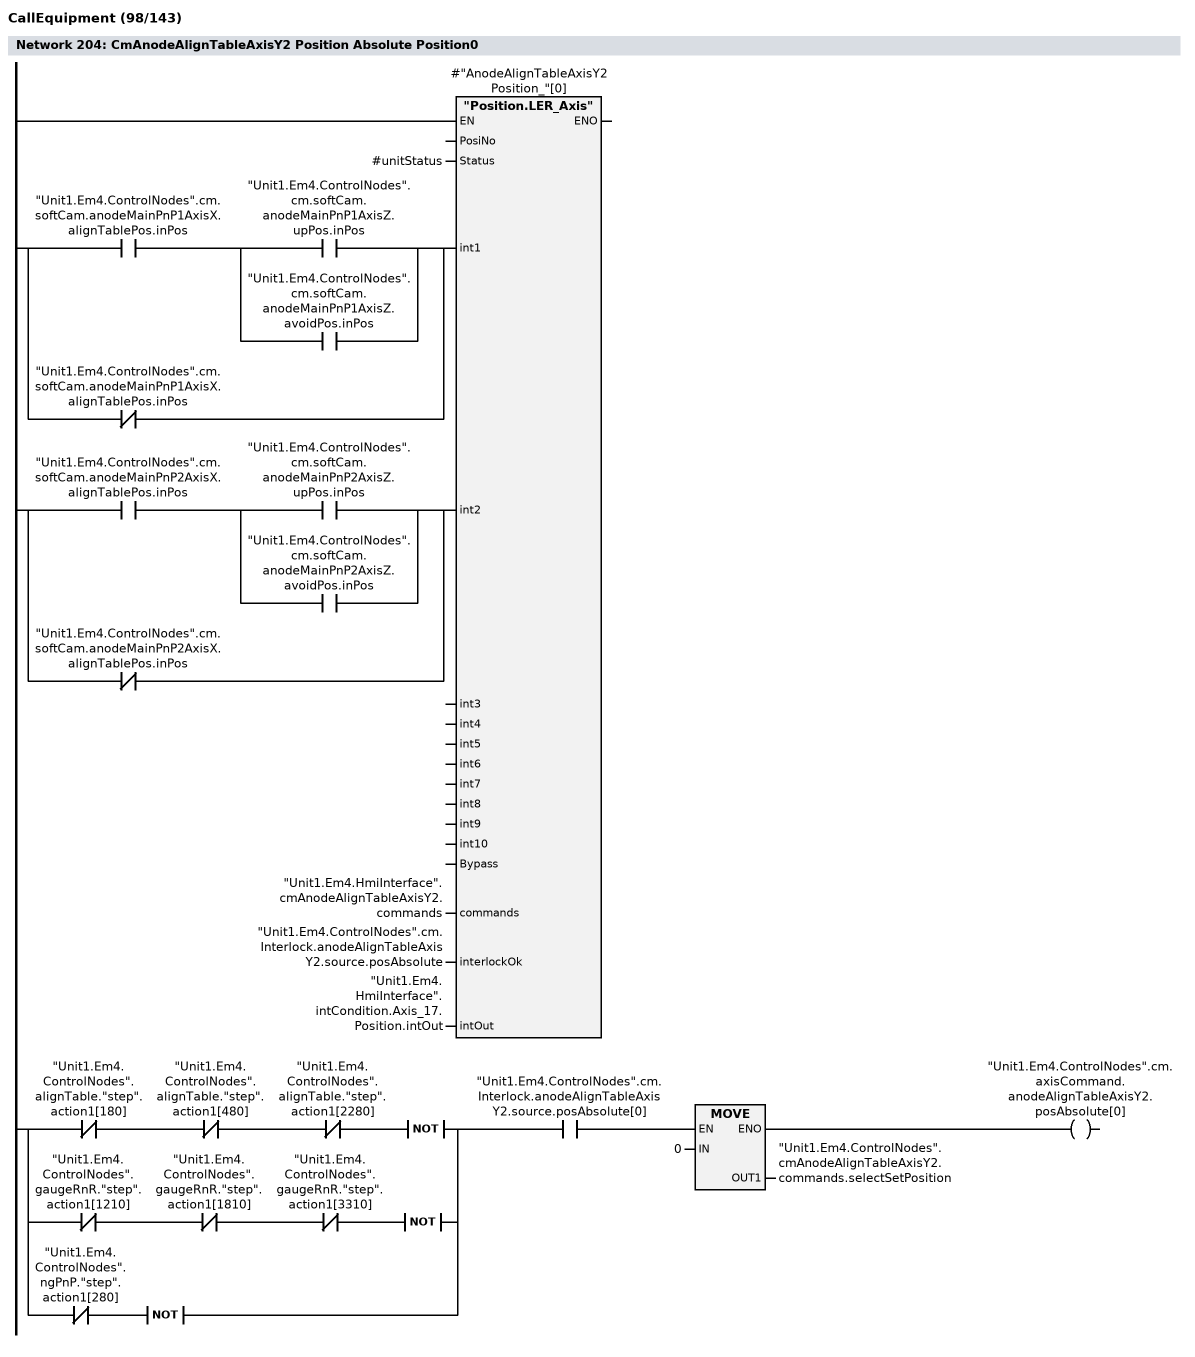
   RUNG wire#powerrail
      #"AnodeAlignTableAxisY2 Position_"[0](int1 := wire#w2, int2 := wire#w4, PosiNo :=, Status := #unitStatus, int3 :=, int4 :=, int5 :=, int6 :=, int7 :=, int8 :=, int9 :=, int10 :=, Bypass :=, commands := "Unit1.Em4.HmiInterface".cmAnodeAlignTableAxisY2.commands, interlockOk := "Unit1.Em4.ControlNodes".cm.Interlock.anodeAlignTableAxisY2.source.posAbsolute, intOut := "Unit1.Em4.HmiInterface".intCondition.Axis_17.Position.intOut)
   END_RUNG
   RUNG wire#powerrail
      Contact( "Unit1.Em4.ControlNodes".cm.softCam.anodeMainPnP1AxisX.alignTablePos.inPos )
      wire#w1
      Contact( "Unit1.Em4.ControlNodes".cm.softCam.anodeMainPnP1AxisZ.upPos.inPos )
   END_RUNG wire#w2
   RUNG wire#w1
      Contact( "Unit1.Em4.ControlNodes".cm.softCam.anodeMainPnP1AxisZ.avoidPos.inPos )
   END_RUNG wire#w2
   RUNG wire#powerrail
      I_Contact( "Unit1.Em4.ControlNodes".cm.softCam.anodeMainPnP1AxisX.alignTablePos.inPos )
   END_RUNG wire#w2
   RUNG wire#powerrail
      Contact( "Unit1.Em4.ControlNodes".cm.softCam.anodeMainPnP2AxisX.alignTablePos.inPos )
      wire#w3
      Contact( "Unit1.Em4.ControlNodes".cm.softCam.anodeMainPnP2AxisZ.upPos.inPos )
   END_RUNG wire#w4
   RUNG wire#w3
      Contact( "Unit1.Em4.ControlNodes".cm.softCam.anodeMainPnP2AxisZ.avoidPos.inPos )
   END_RUNG wire#w4
   RUNG wire#powerrail
      I_Contact( "Unit1.Em4.ControlNodes".cm.softCam.anodeMainPnP2AxisX.alignTablePos.inPos )
   END_RUNG wire#w4
   RUNG wire#powerrail
      I_Contact( "Unit1.Em4.ControlNodes".alignTable."step".action1[180] )
      I_Contact( "Unit1.Em4.ControlNodes".alignTable."step".action1[480] )
      I_Contact( "Unit1.Em4.ControlNodes".alignTable."step".action1[2280] )
      Not()
      wire#w5
      Contact( "Unit1.Em4.ControlNodes".cm.Interlock.anodeAlignTableAxisY2.source.posAbsolute[0] )
      Move(in := 0, out1 => "Unit1.Em4.ControlNodes".cmAnodeAlignTableAxisY2.commands.selectSetPosition)
      Coil( "Unit1.Em4.ControlNodes".cm.axisCommand.anodeAlignTableAxisY2.posAbsolute[0] )
   END_RUNG
   RUNG wire#powerrail
      I_Contact( "Unit1.Em4.ControlNodes".gaugeRnR."step".action1[1210] )
      I_Contact( "Unit1.Em4.ControlNodes".gaugeRnR."step".action1[1810] )
      I_Contact( "Unit1.Em4.ControlNodes".gaugeRnR."step".action1[3310] )
      Not()
   END_RUNG wire#w5
   RUNG wire#powerrail
      I_Contact( "Unit1.Em4.ControlNodes".ngPnP."step".action1[280] )
      Not()
   END_RUNG wire#w5
   // the same network as SCL:
   #"AnodeAlignTableAxisY2 Position_"[0](Status := #unitStatus,   // "Position.LER_Axis"
                           int1 := ("Unit1.Em4.ControlNodes".cm.softCam.anodeMainPnP1AxisX.alignTablePos.inPos AND ("Unit1.Em4.ControlNodes".cm.softCam.anodeMainPnP1AxisZ.upPos.inPos OR "Unit1.Em4.ControlNodes".cm.softCam.anodeMainPnP1AxisZ.avoidPos.inPos)) OR NOT "Unit1.Em4.ControlNodes".cm.softCam.anodeMainPnP1AxisX.alignTablePos.inPos,
                           int2 := ("Unit1.Em4.ControlNodes".cm.softCam.anodeMainPnP2AxisX.alignTablePos.inPos AND ("Unit1.Em4.ControlNodes".cm.softCam.anodeMainPnP2AxisZ.upPos.inPos OR "Unit1.Em4.ControlNodes".cm.softCam.anodeMainPnP2AxisZ.avoidPos.inPos)) OR NOT "Unit1.Em4.ControlNodes".cm.softCam.anodeMainPnP2AxisX.alignTablePos.inPos,
                           commands := "Unit1.Em4.HmiInterface".cmAnodeAlignTableAxisY2.commands,
                           interlockOk := "Unit1.Em4.ControlNodes".cm.Interlock.anodeAlignTableAxisY2.source.posAbsolute,
                           intOut := "Unit1.Em4.HmiInterface".intCondition.Axis_17.Position.intOut);
   #_w1 := (NOT (NOT "Unit1.Em4.ControlNodes".alignTable."step".action1[180] AND NOT "Unit1.Em4.ControlNodes".alignTable."step".action1[480] AND NOT "Unit1.Em4.ControlNodes".alignTable."step".action1[2280]) OR NOT (NOT "Unit1.Em4.ControlNodes".gaugeRnR."step".action1[1210] AND NOT "Unit1.Em4.ControlNodes".gaugeRnR."step".action1[1810] AND NOT "Unit1.Em4.ControlNodes".gaugeRnR."step".action1[3310]) OR NOT (NOT "Unit1.Em4.ControlNodes".ngPnP."step".action1[280])) AND "Unit1.Em4.ControlNodes".cm.Interlock.anodeAlignTableAxisY2.source.posAbsolute[0];
   IF #_w1 THEN "Unit1.Em4.ControlNodes".cmAnodeAlignTableAxisY2.commands.selectSetPosition := 0; END_IF;
   "Unit1.Em4.ControlNodes".cm.axisCommand.anodeAlignTableAxisY2.posAbsolute[0] := #_w1;
END_REGION

REGION Network 205: CmAnodeAlignTableAxisY2 Position Absolute Position1
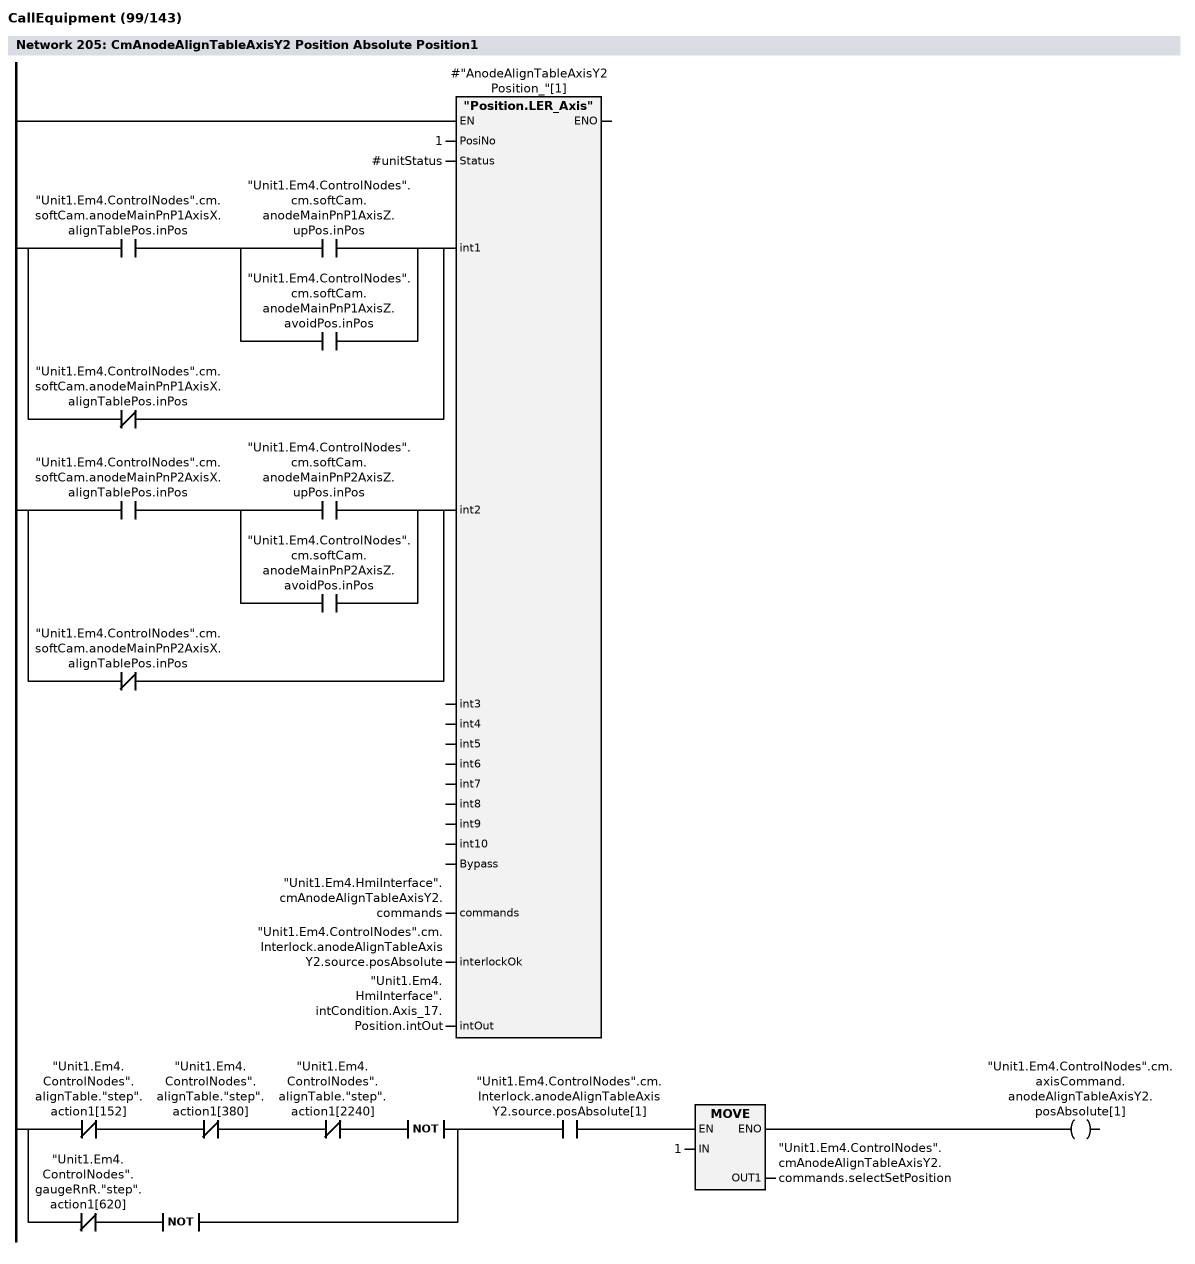
   RUNG wire#powerrail
      #"AnodeAlignTableAxisY2 Position_"[1](int1 := wire#w2, int2 := wire#w4, PosiNo := 1, Status := #unitStatus, int3 :=, int4 :=, int5 :=, int6 :=, int7 :=, int8 :=, int9 :=, int10 :=, Bypass :=, commands := "Unit1.Em4.HmiInterface".cmAnodeAlignTableAxisY2.commands, interlockOk := "Unit1.Em4.ControlNodes".cm.Interlock.anodeAlignTableAxisY2.source.posAbsolute, intOut := "Unit1.Em4.HmiInterface".intCondition.Axis_17.Position.intOut)
   END_RUNG
   RUNG wire#powerrail
      Contact( "Unit1.Em4.ControlNodes".cm.softCam.anodeMainPnP1AxisX.alignTablePos.inPos )
      wire#w1
      Contact( "Unit1.Em4.ControlNodes".cm.softCam.anodeMainPnP1AxisZ.upPos.inPos )
   END_RUNG wire#w2
   RUNG wire#w1
      Contact( "Unit1.Em4.ControlNodes".cm.softCam.anodeMainPnP1AxisZ.avoidPos.inPos )
   END_RUNG wire#w2
   RUNG wire#powerrail
      I_Contact( "Unit1.Em4.ControlNodes".cm.softCam.anodeMainPnP1AxisX.alignTablePos.inPos )
   END_RUNG wire#w2
   RUNG wire#powerrail
      Contact( "Unit1.Em4.ControlNodes".cm.softCam.anodeMainPnP2AxisX.alignTablePos.inPos )
      wire#w3
      Contact( "Unit1.Em4.ControlNodes".cm.softCam.anodeMainPnP2AxisZ.upPos.inPos )
   END_RUNG wire#w4
   RUNG wire#w3
      Contact( "Unit1.Em4.ControlNodes".cm.softCam.anodeMainPnP2AxisZ.avoidPos.inPos )
   END_RUNG wire#w4
   RUNG wire#powerrail
      I_Contact( "Unit1.Em4.ControlNodes".cm.softCam.anodeMainPnP2AxisX.alignTablePos.inPos )
   END_RUNG wire#w4
   RUNG wire#powerrail
      I_Contact( "Unit1.Em4.ControlNodes".alignTable."step".action1[152] )
      I_Contact( "Unit1.Em4.ControlNodes".alignTable."step".action1[380] )
      I_Contact( "Unit1.Em4.ControlNodes".alignTable."step".action1[2240] )
      Not()
      wire#w5
      Contact( "Unit1.Em4.ControlNodes".cm.Interlock.anodeAlignTableAxisY2.source.posAbsolute[1] )
      Move(in := 1, out1 => "Unit1.Em4.ControlNodes".cmAnodeAlignTableAxisY2.commands.selectSetPosition)
      Coil( "Unit1.Em4.ControlNodes".cm.axisCommand.anodeAlignTableAxisY2.posAbsolute[1] )
   END_RUNG
   RUNG wire#powerrail
      I_Contact( "Unit1.Em4.ControlNodes".gaugeRnR."step".action1[620] )
      Not()
   END_RUNG wire#w5
   // the same network as SCL:
   #"AnodeAlignTableAxisY2 Position_"[1](PosiNo := 1,   // "Position.LER_Axis"
                           Status := #unitStatus,
                           int1 := ("Unit1.Em4.ControlNodes".cm.softCam.anodeMainPnP1AxisX.alignTablePos.inPos AND ("Unit1.Em4.ControlNodes".cm.softCam.anodeMainPnP1AxisZ.upPos.inPos OR "Unit1.Em4.ControlNodes".cm.softCam.anodeMainPnP1AxisZ.avoidPos.inPos)) OR NOT "Unit1.Em4.ControlNodes".cm.softCam.anodeMainPnP1AxisX.alignTablePos.inPos,
                           int2 := ("Unit1.Em4.ControlNodes".cm.softCam.anodeMainPnP2AxisX.alignTablePos.inPos AND ("Unit1.Em4.ControlNodes".cm.softCam.anodeMainPnP2AxisZ.upPos.inPos OR "Unit1.Em4.ControlNodes".cm.softCam.anodeMainPnP2AxisZ.avoidPos.inPos)) OR NOT "Unit1.Em4.ControlNodes".cm.softCam.anodeMainPnP2AxisX.alignTablePos.inPos,
                           commands := "Unit1.Em4.HmiInterface".cmAnodeAlignTableAxisY2.commands,
                           interlockOk := "Unit1.Em4.ControlNodes".cm.Interlock.anodeAlignTableAxisY2.source.posAbsolute,
                           intOut := "Unit1.Em4.HmiInterface".intCondition.Axis_17.Position.intOut);
   #_w1 := (NOT (NOT "Unit1.Em4.ControlNodes".alignTable."step".action1[152] AND NOT "Unit1.Em4.ControlNodes".alignTable."step".action1[380] AND NOT "Unit1.Em4.ControlNodes".alignTable."step".action1[2240]) OR NOT (NOT "Unit1.Em4.ControlNodes".gaugeRnR."step".action1[620])) AND "Unit1.Em4.ControlNodes".cm.Interlock.anodeAlignTableAxisY2.source.posAbsolute[1];
   IF #_w1 THEN "Unit1.Em4.ControlNodes".cmAnodeAlignTableAxisY2.commands.selectSetPosition := 1; END_IF;
   "Unit1.Em4.ControlNodes".cm.axisCommand.anodeAlignTableAxisY2.posAbsolute[1] := #_w1;
END_REGION

REGION Network 206: CmAnodeAlignTableAxisY2 Position Absolute Position2
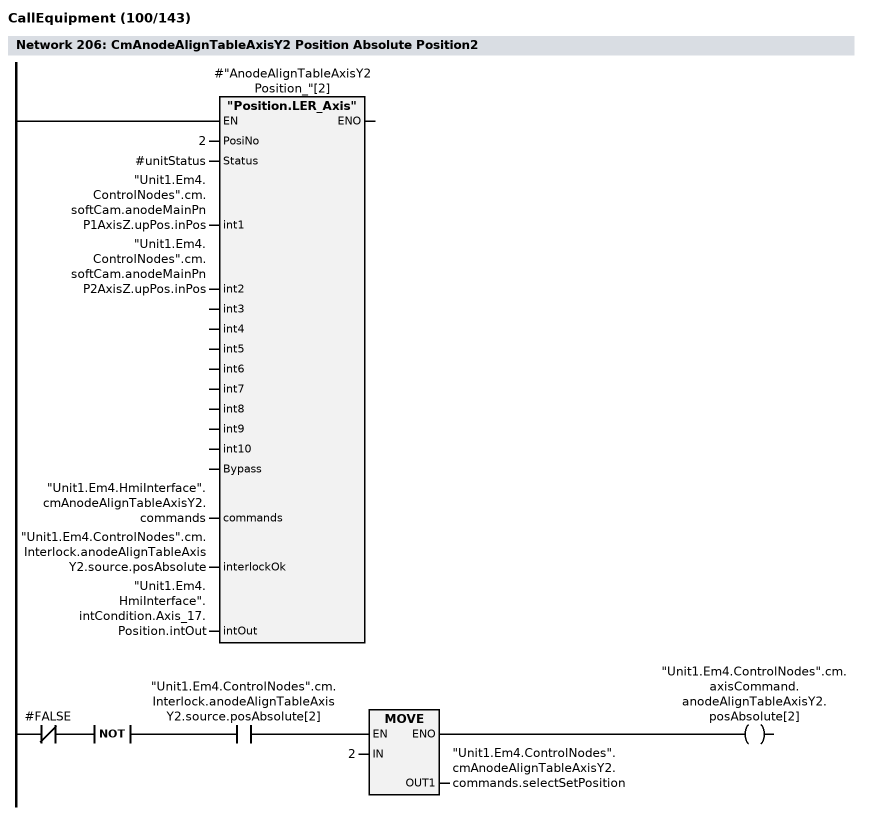
   RUNG wire#powerrail
      #"AnodeAlignTableAxisY2 Position_"[2](PosiNo := 2, Status := #unitStatus, int1 := "Unit1.Em4.ControlNodes".cm.softCam.anodeMainPnP1AxisZ.upPos.inPos, int2 := "Unit1.Em4.ControlNodes".cm.softCam.anodeMainPnP2AxisZ.upPos.inPos, int3 :=, int4 :=, int5 :=, int6 :=, int7 :=, int8 :=, int9 :=, int10 :=, Bypass :=, commands := "Unit1.Em4.HmiInterface".cmAnodeAlignTableAxisY2.commands, interlockOk := "Unit1.Em4.ControlNodes".cm.Interlock.anodeAlignTableAxisY2.source.posAbsolute, intOut := "Unit1.Em4.HmiInterface".intCondition.Axis_17.Position.intOut)
   END_RUNG
   RUNG wire#powerrail
      I_Contact( #FALSE )
      Not()
      Contact( "Unit1.Em4.ControlNodes".cm.Interlock.anodeAlignTableAxisY2.source.posAbsolute[2] )
      Move(in := 2, out1 => "Unit1.Em4.ControlNodes".cmAnodeAlignTableAxisY2.commands.selectSetPosition)
      Coil( "Unit1.Em4.ControlNodes".cm.axisCommand.anodeAlignTableAxisY2.posAbsolute[2] )
   END_RUNG
   // the same network as SCL:
   #"AnodeAlignTableAxisY2 Position_"[2](PosiNo := 2,   // "Position.LER_Axis"
                           Status := #unitStatus,
                           int1 := "Unit1.Em4.ControlNodes".cm.softCam.anodeMainPnP1AxisZ.upPos.inPos,
                           int2 := "Unit1.Em4.ControlNodes".cm.softCam.anodeMainPnP2AxisZ.upPos.inPos,
                           commands := "Unit1.Em4.HmiInterface".cmAnodeAlignTableAxisY2.commands,
                           interlockOk := "Unit1.Em4.ControlNodes".cm.Interlock.anodeAlignTableAxisY2.source.posAbsolute,
                           intOut := "Unit1.Em4.HmiInterface".intCondition.Axis_17.Position.intOut);
   #_w1 := NOT (NOT #FALSE) AND "Unit1.Em4.ControlNodes".cm.Interlock.anodeAlignTableAxisY2.source.posAbsolute[2];
   IF #_w1 THEN "Unit1.Em4.ControlNodes".cmAnodeAlignTableAxisY2.commands.selectSetPosition := 2; END_IF;
   "Unit1.Em4.ControlNodes".cm.axisCommand.anodeAlignTableAxisY2.posAbsolute[2] := #_w1;
END_REGION

REGION Network 207: CmAnodeAlignTableAxisY2 Position Absolute Position3
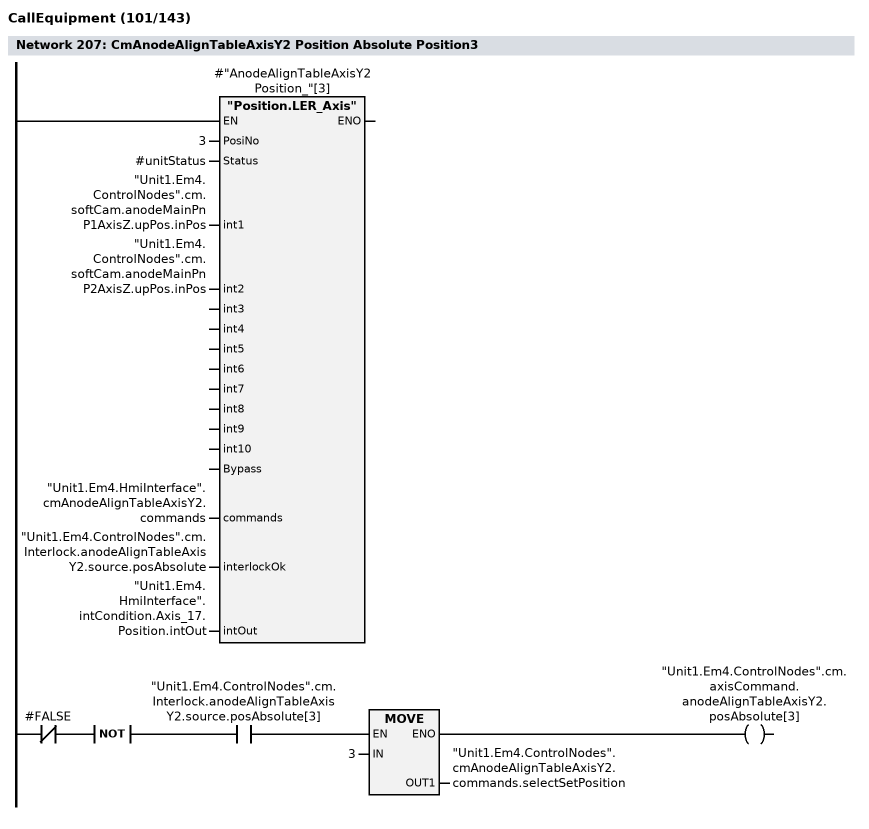
   RUNG wire#powerrail
      #"AnodeAlignTableAxisY2 Position_"[3](PosiNo := 3, Status := #unitStatus, int1 := "Unit1.Em4.ControlNodes".cm.softCam.anodeMainPnP1AxisZ.upPos.inPos, int2 := "Unit1.Em4.ControlNodes".cm.softCam.anodeMainPnP2AxisZ.upPos.inPos, int3 :=, int4 :=, int5 :=, int6 :=, int7 :=, int8 :=, int9 :=, int10 :=, Bypass :=, commands := "Unit1.Em4.HmiInterface".cmAnodeAlignTableAxisY2.commands, interlockOk := "Unit1.Em4.ControlNodes".cm.Interlock.anodeAlignTableAxisY2.source.posAbsolute, intOut := "Unit1.Em4.HmiInterface".intCondition.Axis_17.Position.intOut)
   END_RUNG
   RUNG wire#powerrail
      I_Contact( #FALSE )
      Not()
      Contact( "Unit1.Em4.ControlNodes".cm.Interlock.anodeAlignTableAxisY2.source.posAbsolute[3] )
      Move(in := 3, out1 => "Unit1.Em4.ControlNodes".cmAnodeAlignTableAxisY2.commands.selectSetPosition)
      Coil( "Unit1.Em4.ControlNodes".cm.axisCommand.anodeAlignTableAxisY2.posAbsolute[3] )
   END_RUNG
   // the same network as SCL:
   #"AnodeAlignTableAxisY2 Position_"[3](PosiNo := 3,   // "Position.LER_Axis"
                           Status := #unitStatus,
                           int1 := "Unit1.Em4.ControlNodes".cm.softCam.anodeMainPnP1AxisZ.upPos.inPos,
                           int2 := "Unit1.Em4.ControlNodes".cm.softCam.anodeMainPnP2AxisZ.upPos.inPos,
                           commands := "Unit1.Em4.HmiInterface".cmAnodeAlignTableAxisY2.commands,
                           interlockOk := "Unit1.Em4.ControlNodes".cm.Interlock.anodeAlignTableAxisY2.source.posAbsolute,
                           intOut := "Unit1.Em4.HmiInterface".intCondition.Axis_17.Position.intOut);
   #_w1 := NOT (NOT #FALSE) AND "Unit1.Em4.ControlNodes".cm.Interlock.anodeAlignTableAxisY2.source.posAbsolute[3];
   IF #_w1 THEN "Unit1.Em4.ControlNodes".cmAnodeAlignTableAxisY2.commands.selectSetPosition := 3; END_IF;
   "Unit1.Em4.ControlNodes".cm.axisCommand.anodeAlignTableAxisY2.posAbsolute[3] := #_w1;
END_REGION

REGION Network 208: CmAnodeAlignTableAxisY2 Position Absolute Position4
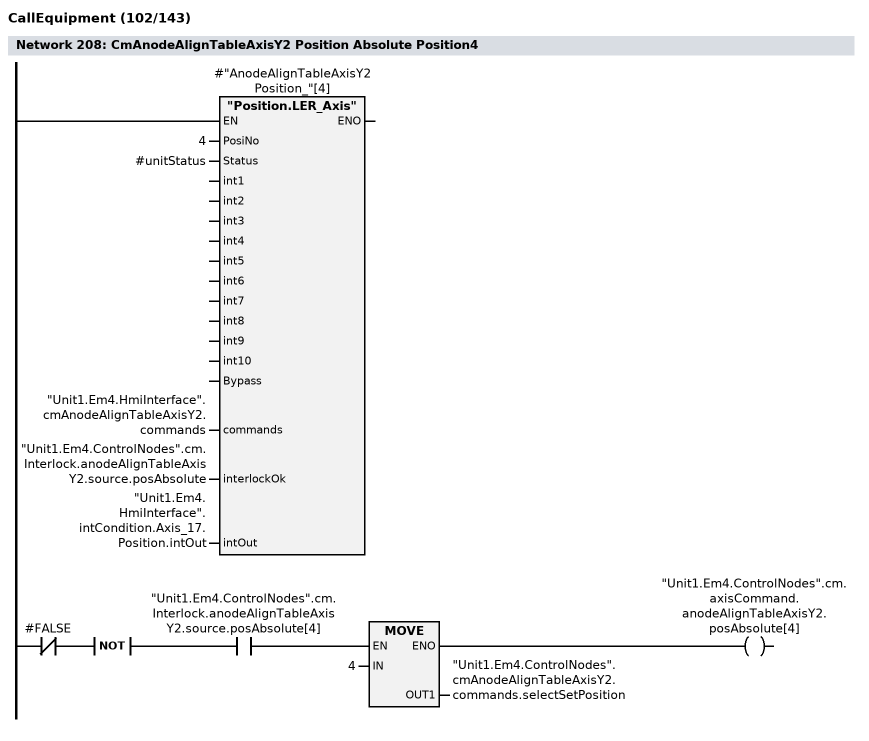
   RUNG wire#powerrail
      #"AnodeAlignTableAxisY2 Position_"[4](PosiNo := 4, Status := #unitStatus, int1 :=, int2 :=, int3 :=, int4 :=, int5 :=, int6 :=, int7 :=, int8 :=, int9 :=, int10 :=, Bypass :=, commands := "Unit1.Em4.HmiInterface".cmAnodeAlignTableAxisY2.commands, interlockOk := "Unit1.Em4.ControlNodes".cm.Interlock.anodeAlignTableAxisY2.source.posAbsolute, intOut := "Unit1.Em4.HmiInterface".intCondition.Axis_17.Position.intOut)
   END_RUNG
   RUNG wire#powerrail
      I_Contact( #FALSE )
      Not()
      Contact( "Unit1.Em4.ControlNodes".cm.Interlock.anodeAlignTableAxisY2.source.posAbsolute[4] )
      Move(in := 4, out1 => "Unit1.Em4.ControlNodes".cmAnodeAlignTableAxisY2.commands.selectSetPosition)
      Coil( "Unit1.Em4.ControlNodes".cm.axisCommand.anodeAlignTableAxisY2.posAbsolute[4] )
   END_RUNG
   // the same network as SCL:
   #"AnodeAlignTableAxisY2 Position_"[4](PosiNo := 4,   // "Position.LER_Axis"
                           Status := #unitStatus,
                           commands := "Unit1.Em4.HmiInterface".cmAnodeAlignTableAxisY2.commands,
                           interlockOk := "Unit1.Em4.ControlNodes".cm.Interlock.anodeAlignTableAxisY2.source.posAbsolute,
                           intOut := "Unit1.Em4.HmiInterface".intCondition.Axis_17.Position.intOut);
   #_w1 := NOT (NOT #FALSE) AND "Unit1.Em4.ControlNodes".cm.Interlock.anodeAlignTableAxisY2.source.posAbsolute[4];
   IF #_w1 THEN "Unit1.Em4.ControlNodes".cmAnodeAlignTableAxisY2.commands.selectSetPosition := 4; END_IF;
   "Unit1.Em4.ControlNodes".cm.axisCommand.anodeAlignTableAxisY2.posAbsolute[4] := #_w1;
END_REGION

REGION Network 209: CmAnodeAlignTableAxisY2 Position Absolute Position5
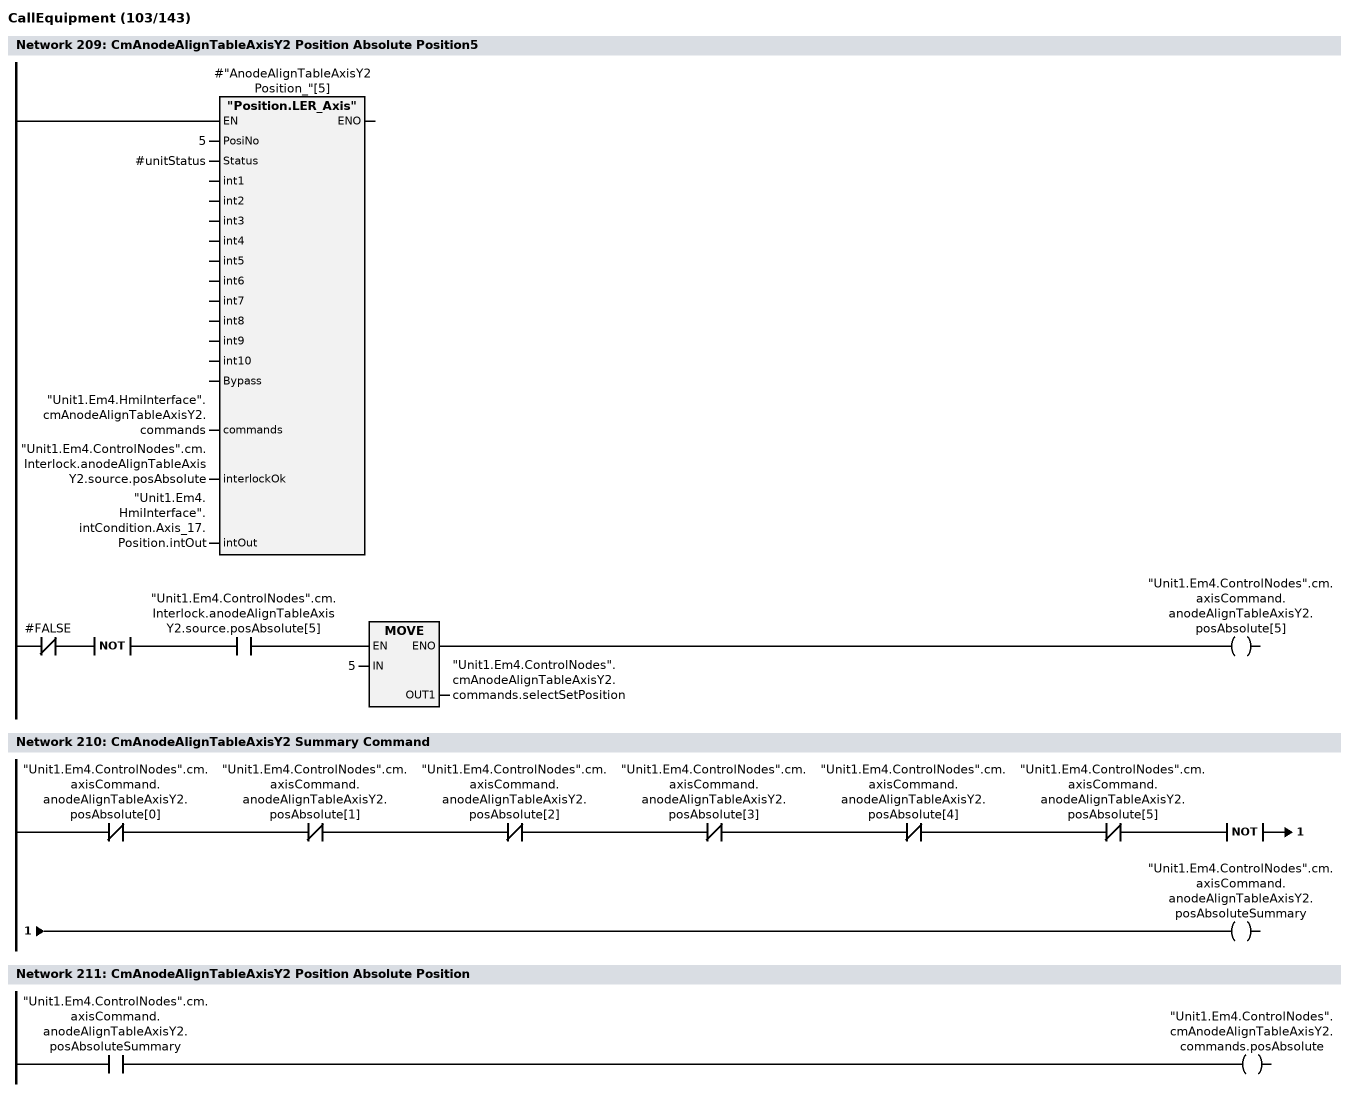
   RUNG wire#powerrail
      #"AnodeAlignTableAxisY2 Position_"[5](PosiNo := 5, Status := #unitStatus, int1 :=, int2 :=, int3 :=, int4 :=, int5 :=, int6 :=, int7 :=, int8 :=, int9 :=, int10 :=, Bypass :=, commands := "Unit1.Em4.HmiInterface".cmAnodeAlignTableAxisY2.commands, interlockOk := "Unit1.Em4.ControlNodes".cm.Interlock.anodeAlignTableAxisY2.source.posAbsolute, intOut := "Unit1.Em4.HmiInterface".intCondition.Axis_17.Position.intOut)
   END_RUNG
   RUNG wire#powerrail
      I_Contact( #FALSE )
      Not()
      Contact( "Unit1.Em4.ControlNodes".cm.Interlock.anodeAlignTableAxisY2.source.posAbsolute[5] )
      Move(in := 5, out1 => "Unit1.Em4.ControlNodes".cmAnodeAlignTableAxisY2.commands.selectSetPosition)
      Coil( "Unit1.Em4.ControlNodes".cm.axisCommand.anodeAlignTableAxisY2.posAbsolute[5] )
   END_RUNG
   // the same network as SCL:
   #"AnodeAlignTableAxisY2 Position_"[5](PosiNo := 5,   // "Position.LER_Axis"
                           Status := #unitStatus,
                           commands := "Unit1.Em4.HmiInterface".cmAnodeAlignTableAxisY2.commands,
                           interlockOk := "Unit1.Em4.ControlNodes".cm.Interlock.anodeAlignTableAxisY2.source.posAbsolute,
                           intOut := "Unit1.Em4.HmiInterface".intCondition.Axis_17.Position.intOut);
   #_w1 := NOT (NOT #FALSE) AND "Unit1.Em4.ControlNodes".cm.Interlock.anodeAlignTableAxisY2.source.posAbsolute[5];
   IF #_w1 THEN "Unit1.Em4.ControlNodes".cmAnodeAlignTableAxisY2.commands.selectSetPosition := 5; END_IF;
   "Unit1.Em4.ControlNodes".cm.axisCommand.anodeAlignTableAxisY2.posAbsolute[5] := #_w1;
END_REGION

REGION Network 210: CmAnodeAlignTableAxisY2 Summary Command
   RUNG wire#powerrail
      I_Contact( "Unit1.Em4.ControlNodes".cm.axisCommand.anodeAlignTableAxisY2.posAbsolute[0] )
      I_Contact( "Unit1.Em4.ControlNodes".cm.axisCommand.anodeAlignTableAxisY2.posAbsolute[1] )
      I_Contact( "Unit1.Em4.ControlNodes".cm.axisCommand.anodeAlignTableAxisY2.posAbsolute[2] )
      I_Contact( "Unit1.Em4.ControlNodes".cm.axisCommand.anodeAlignTableAxisY2.posAbsolute[3] )
      I_Contact( "Unit1.Em4.ControlNodes".cm.axisCommand.anodeAlignTableAxisY2.posAbsolute[4] )
      I_Contact( "Unit1.Em4.ControlNodes".cm.axisCommand.anodeAlignTableAxisY2.posAbsolute[5] )
      Not()
      Coil( "Unit1.Em4.ControlNodes".cm.axisCommand.anodeAlignTableAxisY2.posAbsoluteSummary )
   END_RUNG
   // the same network as SCL:
   "Unit1.Em4.ControlNodes".cm.axisCommand.anodeAlignTableAxisY2.posAbsoluteSummary := NOT (NOT "Unit1.Em4.ControlNodes".cm.axisCommand.anodeAlignTableAxisY2.posAbsolute[0] AND NOT "Unit1.Em4.ControlNodes".cm.axisCommand.anodeAlignTableAxisY2.posAbsolute[1] AND NOT "Unit1.Em4.ControlNodes".cm.axisCommand.anodeAlignTableAxisY2.posAbsolute[2] AND NOT "Unit1.Em4.ControlNodes".cm.axisCommand.anodeAlignTableAxisY2.posAbsolute[3] AND NOT "Unit1.Em4.ControlNodes".cm.axisCommand.anodeAlignTableAxisY2.posAbsolute[4] AND NOT "Unit1.Em4.ControlNodes".cm.axisCommand.anodeAlignTableAxisY2.posAbsolute[5]);
END_REGION

REGION Network 211: CmAnodeAlignTableAxisY2 Position Absolute Position
   RUNG wire#powerrail
      Contact( "Unit1.Em4.ControlNodes".cm.axisCommand.anodeAlignTableAxisY2.posAbsoluteSummary )
      Coil( "Unit1.Em4.ControlNodes".cmAnodeAlignTableAxisY2.commands.posAbsolute )
   END_RUNG
   // the same network as SCL:
   "Unit1.Em4.ControlNodes".cmAnodeAlignTableAxisY2.commands.posAbsolute := "Unit1.Em4.ControlNodes".cm.axisCommand.anodeAlignTableAxisY2.posAbsoluteSummary;
END_REGION

REGION Network 212: CmAnodeAlignTableAxisY1 Interlock Summary
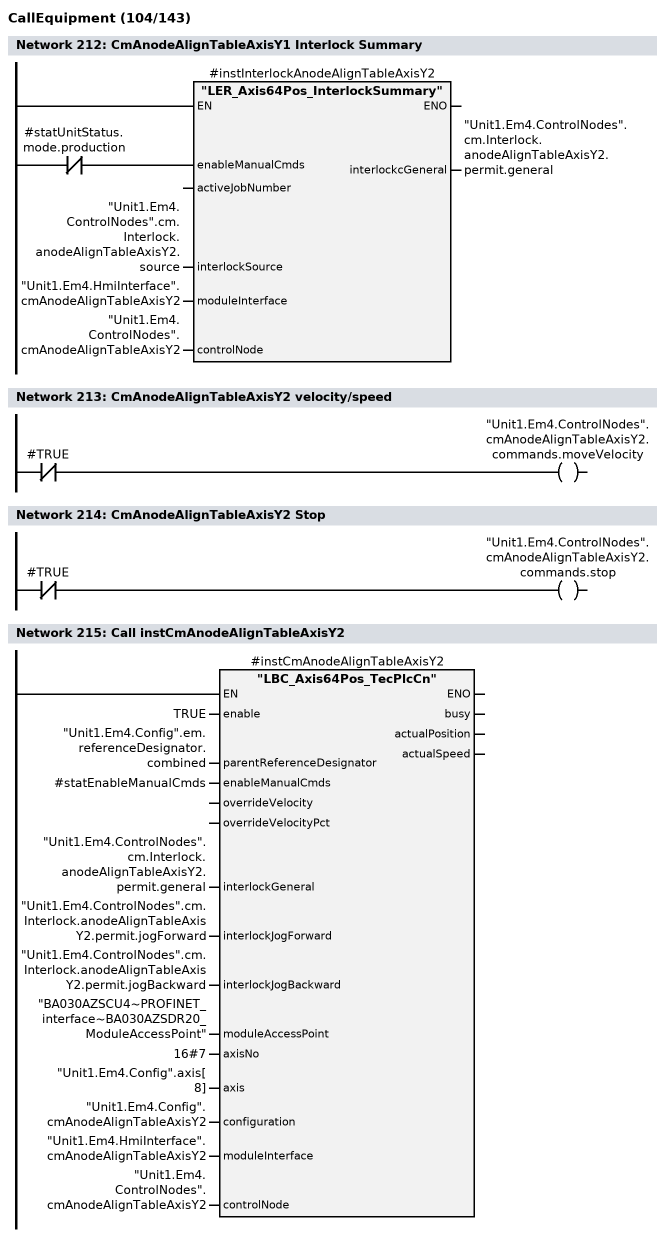
   RUNG wire#powerrail
      #instInterlockAnodeAlignTableAxisY2(enableManualCmds := wire#w1, activeJobNumber :=, interlockSource := "Unit1.Em4.ControlNodes".cm.Interlock.anodeAlignTableAxisY2.source, moduleInterface := "Unit1.Em4.HmiInterface".cmAnodeAlignTableAxisY2, controlNode := "Unit1.Em4.ControlNodes".cmAnodeAlignTableAxisY2, interlockcGeneral => "Unit1.Em4.ControlNodes".cm.Interlock.anodeAlignTableAxisY2.permit.general)
   END_RUNG
   RUNG wire#powerrail
      I_Contact( #statUnitStatus.mode.production )
   END_RUNG wire#w1
   // the same network as SCL:
   #instInterlockAnodeAlignTableAxisY2(enableManualCmds := NOT #statUnitStatus.mode.production,   // "LER_Axis64Pos_InterlockSummary"
                           interlockSource := "Unit1.Em4.ControlNodes".cm.Interlock.anodeAlignTableAxisY2.source,
                           moduleInterface := "Unit1.Em4.HmiInterface".cmAnodeAlignTableAxisY2,
                           controlNode := "Unit1.Em4.ControlNodes".cmAnodeAlignTableAxisY2,
                           interlockcGeneral => "Unit1.Em4.ControlNodes".cm.Interlock.anodeAlignTableAxisY2.permit.general);
END_REGION

REGION Network 213: CmAnodeAlignTableAxisY2 velocity/speed
   RUNG wire#powerrail
      I_Contact( #TRUE )
      Coil( "Unit1.Em4.ControlNodes".cmAnodeAlignTableAxisY2.commands.moveVelocity )
   END_RUNG
   // the same network as SCL:
   "Unit1.Em4.ControlNodes".cmAnodeAlignTableAxisY2.commands.moveVelocity := NOT #TRUE;
END_REGION

REGION Network 214: CmAnodeAlignTableAxisY2 Stop
   RUNG wire#powerrail
      I_Contact( #TRUE )
      Coil( "Unit1.Em4.ControlNodes".cmAnodeAlignTableAxisY2.commands.stop )
   END_RUNG
   // the same network as SCL:
   "Unit1.Em4.ControlNodes".cmAnodeAlignTableAxisY2.commands.stop := NOT #TRUE;
END_REGION

REGION Network 215: Call instCmAnodeAlignTableAxisY2
   RUNG wire#powerrail
      #instCmAnodeAlignTableAxisY2(enable := TRUE, parentReferenceDesignator := "Unit1.Em4.Config".em.referenceDesignator.combined, enableManualCmds := #statEnableManualCmds, overrideVelocity :=, overrideVelocityPct :=, interlockGeneral := "Unit1.Em4.ControlNodes".cm.Interlock.anodeAlignTableAxisY2.permit.general, interlockJogForward := "Unit1.Em4.ControlNodes".cm.Interlock.anodeAlignTableAxisY2.permit.jogForward, interlockJogBackward := "Unit1.Em4.ControlNodes".cm.Interlock.anodeAlignTableAxisY2.permit.jogBackward, moduleAccessPoint := "BA030AZSCU4~PROFINET_interface~BA030AZSDR20_ModuleAccessPoint", axisNo := 16#7, axis := "Unit1.Em4.Config".axis[8], configuration := "Unit1.Em4.Config".cmAnodeAlignTableAxisY2, moduleInterface := "Unit1.Em4.HmiInterface".cmAnodeAlignTableAxisY2, controlNode := "Unit1.Em4.ControlNodes".cmAnodeAlignTableAxisY2, busy =>, actualPosition =>, actualSpeed =>)
   END_RUNG
   // the same network as SCL:
   #instCmAnodeAlignTableAxisY2(enable := TRUE,   // "LBC_Axis64Pos_TecPlcCn"
                           parentReferenceDesignator := "Unit1.Em4.Config".em.referenceDesignator.combined,
                           enableManualCmds := #statEnableManualCmds,
                           interlockGeneral := "Unit1.Em4.ControlNodes".cm.Interlock.anodeAlignTableAxisY2.permit.general,
                           interlockJogForward := "Unit1.Em4.ControlNodes".cm.Interlock.anodeAlignTableAxisY2.permit.jogForward,
                           interlockJogBackward := "Unit1.Em4.ControlNodes".cm.Interlock.anodeAlignTableAxisY2.permit.jogBackward,
                           moduleAccessPoint := "BA030AZSCU4~PROFINET_interface~BA030AZSDR20_ModuleAccessPoint",
                           axisNo := 16#7,
                           axis := "Unit1.Em4.Config".axis[8],
                           configuration := "Unit1.Em4.Config".cmAnodeAlignTableAxisY2,
                           moduleInterface := "Unit1.Em4.HmiInterface".cmAnodeAlignTableAxisY2,
                           controlNode := "Unit1.Em4.ControlNodes".cmAnodeAlignTableAxisY2);
END_REGION

REGION Network 216: AnodeAlignTableAxisY1 SoftCam
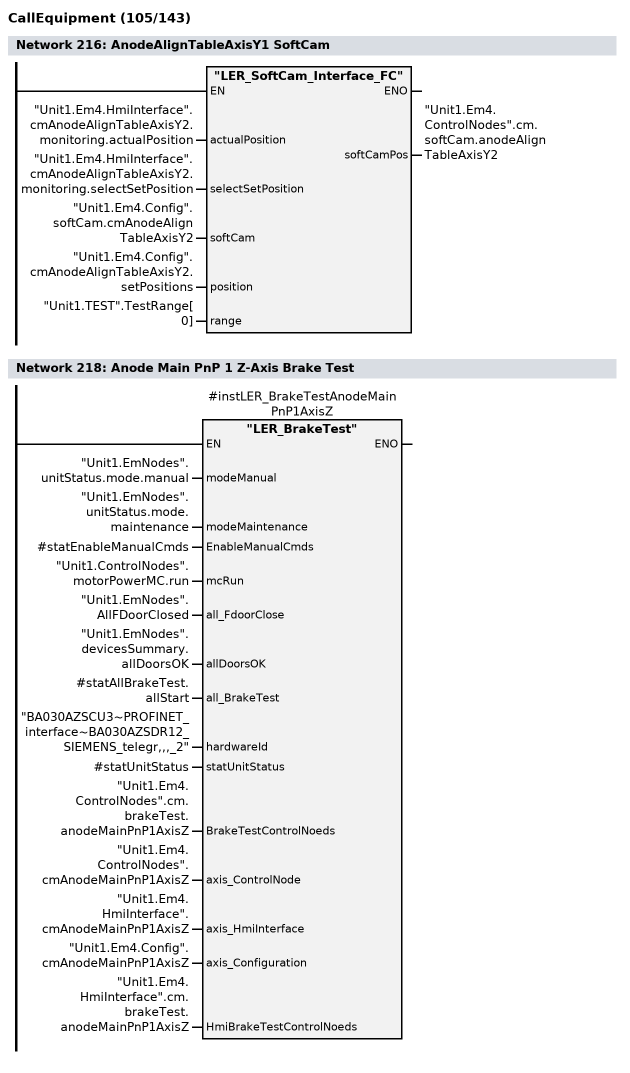
   RUNG wire#powerrail
      "LER_SoftCam_Interface_FC"(actualPosition := "Unit1.Em4.HmiInterface".cmAnodeAlignTableAxisY2.monitoring.actualPosition, selectSetPosition := "Unit1.Em4.HmiInterface".cmAnodeAlignTableAxisY2.monitoring.selectSetPosition, softCam := "Unit1.Em4.Config".softCam.cmAnodeAlignTableAxisY2, position := "Unit1.Em4.Config".cmAnodeAlignTableAxisY2.setPositions, range := "Unit1.TEST".TestRange[0], softCamPos => "Unit1.Em4.ControlNodes".cm.softCam.anodeAlignTableAxisY2)
   END_RUNG
   // the same network as SCL:
   "LER_SoftCam_Interface_FC"(actualPosition := "Unit1.Em4.HmiInterface".cmAnodeAlignTableAxisY2.monitoring.actualPosition,
                           selectSetPosition := "Unit1.Em4.HmiInterface".cmAnodeAlignTableAxisY2.monitoring.selectSetPosition,
                           softCam := "Unit1.Em4.Config".softCam.cmAnodeAlignTableAxisY2,
                           position := "Unit1.Em4.Config".cmAnodeAlignTableAxisY2.setPositions,
                           range := "Unit1.TEST".TestRange[0],
                           softCamPos => "Unit1.Em4.ControlNodes".cm.softCam.anodeAlignTableAxisY2);
END_REGION

REGION Network 217: ******************** Brake Test (Axis) ********************
END_REGION

REGION Network 218: Anode Main PnP 1 Z-Axis Brake Test
   RUNG wire#powerrail
      #instLER_BrakeTestAnodeMainPnP1AxisZ(modeManual := "Unit1.EmNodes".unitStatus.mode.manual, modeMaintenance := "Unit1.EmNodes".unitStatus.mode.maintenance, EnableManualCmds := #statEnableManualCmds, mcRun := "Unit1.ControlNodes".motorPowerMC.run, all_FdoorClose := "Unit1.EmNodes".AllFDoorClosed, allDoorsOK := "Unit1.EmNodes".devicesSummary.allDoorsOK, all_BrakeTest := #statAllBrakeTest.allStart, hardwareId := "BA030AZSCU3~PROFINET_interface~BA030AZSDR12_SIEMENS_telegr,,,_2", statUnitStatus := #statUnitStatus, BrakeTestControlNoeds := "Unit1.Em4.ControlNodes".cm.brakeTest.anodeMainPnP1AxisZ, axis_ControlNode := "Unit1.Em4.ControlNodes".cmAnodeMainPnP1AxisZ, axis_HmiInterface := "Unit1.Em4.HmiInterface".cmAnodeMainPnP1AxisZ, axis_Configuration := "Unit1.Em4.Config".cmAnodeMainPnP1AxisZ, HmiBrakeTestControlNoeds := "Unit1.Em4.HmiInterface".cm.brakeTest.anodeMainPnP1AxisZ)
   END_RUNG
   // the same network as SCL:
   #instLER_BrakeTestAnodeMainPnP1AxisZ(modeManual := "Unit1.EmNodes".unitStatus.mode.manual,   // "LER_BrakeTest"
                           modeMaintenance := "Unit1.EmNodes".unitStatus.mode.maintenance,
                           EnableManualCmds := #statEnableManualCmds,
                           mcRun := "Unit1.ControlNodes".motorPowerMC.run,
                           all_FdoorClose := "Unit1.EmNodes".AllFDoorClosed,
                           allDoorsOK := "Unit1.EmNodes".devicesSummary.allDoorsOK,
                           all_BrakeTest := #statAllBrakeTest.allStart,
                           hardwareId := "BA030AZSCU3~PROFINET_interface~BA030AZSDR12_SIEMENS_telegr,,,_2",
                           statUnitStatus := #statUnitStatus,
                           BrakeTestControlNoeds := "Unit1.Em4.ControlNodes".cm.brakeTest.anodeMainPnP1AxisZ,
                           axis_ControlNode := "Unit1.Em4.ControlNodes".cmAnodeMainPnP1AxisZ,
                           axis_HmiInterface := "Unit1.Em4.HmiInterface".cmAnodeMainPnP1AxisZ,
                           axis_Configuration := "Unit1.Em4.Config".cmAnodeMainPnP1AxisZ,
                           HmiBrakeTestControlNoeds := "Unit1.Em4.HmiInterface".cm.brakeTest.anodeMainPnP1AxisZ);
END_REGION

REGION Network 219: Anode Main PnP 2 Z-Axis Brake Test
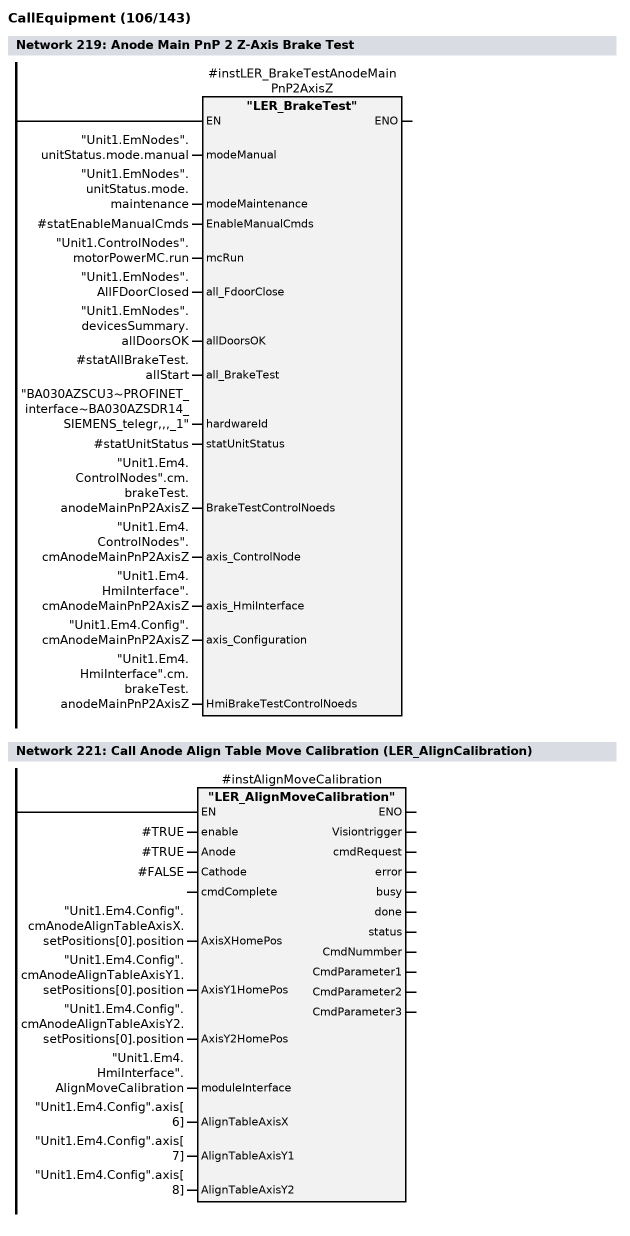
   RUNG wire#powerrail
      #instLER_BrakeTestAnodeMainPnP2AxisZ(modeManual := "Unit1.EmNodes".unitStatus.mode.manual, modeMaintenance := "Unit1.EmNodes".unitStatus.mode.maintenance, EnableManualCmds := #statEnableManualCmds, mcRun := "Unit1.ControlNodes".motorPowerMC.run, all_FdoorClose := "Unit1.EmNodes".AllFDoorClosed, allDoorsOK := "Unit1.EmNodes".devicesSummary.allDoorsOK, all_BrakeTest := #statAllBrakeTest.allStart, hardwareId := "BA030AZSCU3~PROFINET_interface~BA030AZSDR14_SIEMENS_telegr,,,_1", statUnitStatus := #statUnitStatus, BrakeTestControlNoeds := "Unit1.Em4.ControlNodes".cm.brakeTest.anodeMainPnP2AxisZ, axis_ControlNode := "Unit1.Em4.ControlNodes".cmAnodeMainPnP2AxisZ, axis_HmiInterface := "Unit1.Em4.HmiInterface".cmAnodeMainPnP2AxisZ, axis_Configuration := "Unit1.Em4.Config".cmAnodeMainPnP2AxisZ, HmiBrakeTestControlNoeds := "Unit1.Em4.HmiInterface".cm.brakeTest.anodeMainPnP2AxisZ)
   END_RUNG
   // the same network as SCL:
   #instLER_BrakeTestAnodeMainPnP2AxisZ(modeManual := "Unit1.EmNodes".unitStatus.mode.manual,   // "LER_BrakeTest"
                           modeMaintenance := "Unit1.EmNodes".unitStatus.mode.maintenance,
                           EnableManualCmds := #statEnableManualCmds,
                           mcRun := "Unit1.ControlNodes".motorPowerMC.run,
                           all_FdoorClose := "Unit1.EmNodes".AllFDoorClosed,
                           allDoorsOK := "Unit1.EmNodes".devicesSummary.allDoorsOK,
                           all_BrakeTest := #statAllBrakeTest.allStart,
                           hardwareId := "BA030AZSCU3~PROFINET_interface~BA030AZSDR14_SIEMENS_telegr,,,_1",
                           statUnitStatus := #statUnitStatus,
                           BrakeTestControlNoeds := "Unit1.Em4.ControlNodes".cm.brakeTest.anodeMainPnP2AxisZ,
                           axis_ControlNode := "Unit1.Em4.ControlNodes".cmAnodeMainPnP2AxisZ,
                           axis_HmiInterface := "Unit1.Em4.HmiInterface".cmAnodeMainPnP2AxisZ,
                           axis_Configuration := "Unit1.Em4.Config".cmAnodeMainPnP2AxisZ,
                           HmiBrakeTestControlNoeds := "Unit1.Em4.HmiInterface".cm.brakeTest.anodeMainPnP2AxisZ);
END_REGION

REGION Network 220: ******************** Align Table Extended Function ********************
END_REGION

REGION Network 221: Call Anode Align Table Move Calibration (LER_AlignCalibration)
   RUNG wire#powerrail
      #instAlignMoveCalibration(enable := #TRUE, Anode := #TRUE, Cathode := #FALSE, cmdComplete :=, AxisXHomePos := "Unit1.Em4.Config".cmAnodeAlignTableAxisX.setPositions[0].position, AxisY1HomePos := "Unit1.Em4.Config".cmAnodeAlignTableAxisY1.setPositions[0].position, AxisY2HomePos := "Unit1.Em4.Config".cmAnodeAlignTableAxisY2.setPositions[0].position, moduleInterface := "Unit1.Em4.HmiInterface".AlignMoveCalibration, AlignTableAxisX := "Unit1.Em4.Config".axis[6], AlignTableAxisY1 := "Unit1.Em4.Config".axis[7], AlignTableAxisY2 := "Unit1.Em4.Config".axis[8], Visiontrigger =>, cmdRequest =>, error =>, busy =>, done =>, status =>, CmdNummber =>, CmdParameter1 =>, CmdParameter2 =>, CmdParameter3 =>)
   END_RUNG
   // the same network as SCL:
   #instAlignMoveCalibration(enable := #TRUE,   // "LER_AlignMoveCalibration"
                           Anode := #TRUE,
                           Cathode := #FALSE,
                           AxisXHomePos := "Unit1.Em4.Config".cmAnodeAlignTableAxisX.setPositions[0].position,
                           AxisY1HomePos := "Unit1.Em4.Config".cmAnodeAlignTableAxisY1.setPositions[0].position,
                           AxisY2HomePos := "Unit1.Em4.Config".cmAnodeAlignTableAxisY2.setPositions[0].position,
                           moduleInterface := "Unit1.Em4.HmiInterface".AlignMoveCalibration,
                           AlignTableAxisX := "Unit1.Em4.Config".axis[6],
                           AlignTableAxisY1 := "Unit1.Em4.Config".axis[7],
                           AlignTableAxisY2 := "Unit1.Em4.Config".axis[8]);
END_REGION

REGION Network 222: Call Anode Align Table Theta Calibration (LER_AlignCalibration)
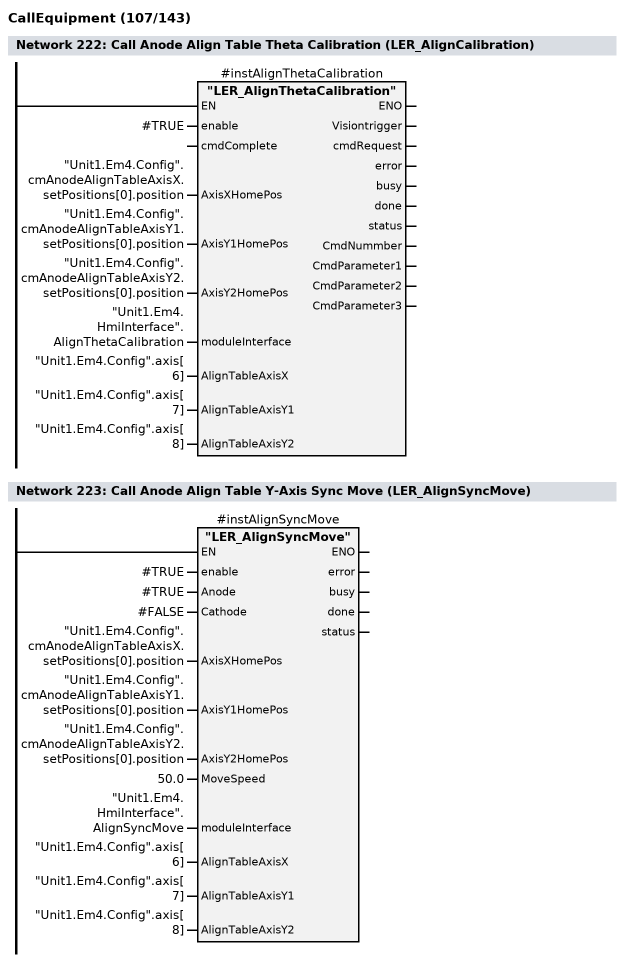
   RUNG wire#powerrail
      #instAlignThetaCalibration(enable := #TRUE, cmdComplete :=, AxisXHomePos := "Unit1.Em4.Config".cmAnodeAlignTableAxisX.setPositions[0].position, AxisY1HomePos := "Unit1.Em4.Config".cmAnodeAlignTableAxisY1.setPositions[0].position, AxisY2HomePos := "Unit1.Em4.Config".cmAnodeAlignTableAxisY2.setPositions[0].position, moduleInterface := "Unit1.Em4.HmiInterface".AlignThetaCalibration, AlignTableAxisX := "Unit1.Em4.Config".axis[6], AlignTableAxisY1 := "Unit1.Em4.Config".axis[7], AlignTableAxisY2 := "Unit1.Em4.Config".axis[8], Visiontrigger =>, cmdRequest =>, error =>, busy =>, done =>, status =>, CmdNummber =>, CmdParameter1 =>, CmdParameter2 =>, CmdParameter3 =>)
   END_RUNG
   // the same network as SCL:
   #instAlignThetaCalibration(enable := #TRUE,   // "LER_AlignThetaCalibration"
                           AxisXHomePos := "Unit1.Em4.Config".cmAnodeAlignTableAxisX.setPositions[0].position,
                           AxisY1HomePos := "Unit1.Em4.Config".cmAnodeAlignTableAxisY1.setPositions[0].position,
                           AxisY2HomePos := "Unit1.Em4.Config".cmAnodeAlignTableAxisY2.setPositions[0].position,
                           moduleInterface := "Unit1.Em4.HmiInterface".AlignThetaCalibration,
                           AlignTableAxisX := "Unit1.Em4.Config".axis[6],
                           AlignTableAxisY1 := "Unit1.Em4.Config".axis[7],
                           AlignTableAxisY2 := "Unit1.Em4.Config".axis[8]);
END_REGION

REGION Network 223: Call Anode Align Table Y-Axis Sync Move (LER_AlignSyncMove)
   RUNG wire#powerrail
      #instAlignSyncMove(enable := #TRUE, Anode := #TRUE, Cathode := #FALSE, AxisXHomePos := "Unit1.Em4.Config".cmAnodeAlignTableAxisX.setPositions[0].position, AxisY1HomePos := "Unit1.Em4.Config".cmAnodeAlignTableAxisY1.setPositions[0].position, AxisY2HomePos := "Unit1.Em4.Config".cmAnodeAlignTableAxisY2.setPositions[0].position, MoveSpeed := 50.0, moduleInterface := "Unit1.Em4.HmiInterface".AlignSyncMove, AlignTableAxisX := "Unit1.Em4.Config".axis[6], AlignTableAxisY1 := "Unit1.Em4.Config".axis[7], AlignTableAxisY2 := "Unit1.Em4.Config".axis[8], error =>, busy =>, done =>, status =>)
   END_RUNG
   // the same network as SCL:
   #instAlignSyncMove(enable := #TRUE,   // "LER_AlignSyncMove"
                      Anode := #TRUE,
                      Cathode := #FALSE,
                      AxisXHomePos := "Unit1.Em4.Config".cmAnodeAlignTableAxisX.setPositions[0].position,
                      AxisY1HomePos := "Unit1.Em4.Config".cmAnodeAlignTableAxisY1.setPositions[0].position,
                      AxisY2HomePos := "Unit1.Em4.Config".cmAnodeAlignTableAxisY2.setPositions[0].position,
                      MoveSpeed := 50.0,
                      moduleInterface := "Unit1.Em4.HmiInterface".AlignSyncMove,
                      AlignTableAxisX := "Unit1.Em4.Config".axis[6],
                      AlignTableAxisY1 := "Unit1.Em4.Config".axis[7],
                      AlignTableAxisY2 := "Unit1.Em4.Config".axis[8]);
END_REGION

REGION Network 224: ********** Control Modules (TwoWayActuator) **********
END_REGION

REGION Network 225: Reset CMS
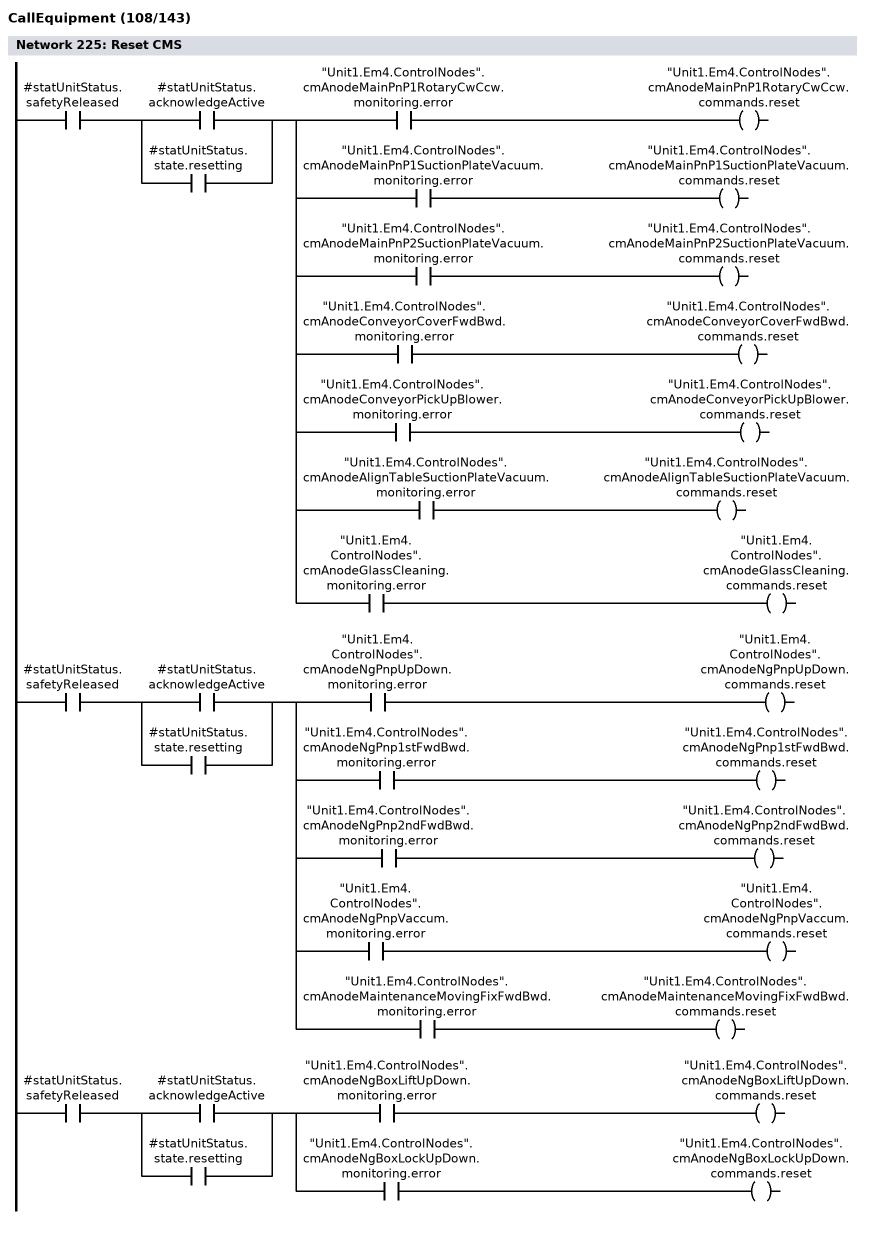
   RUNG wire#powerrail
      Contact( #statUnitStatus.safetyReleased )
      wire#w1
      Contact( #statUnitStatus.acknowledgeActive )
      wire#w2
      Contact( "Unit1.Em4.ControlNodes".cmAnodeMainPnP1RotaryCwCcw.monitoring.error )
      Coil( "Unit1.Em4.ControlNodes".cmAnodeMainPnP1RotaryCwCcw.commands.reset )
   END_RUNG
   RUNG wire#w1
      Contact( #statUnitStatus.state.resetting )
   END_RUNG wire#w2
   RUNG wire#w2
      Contact( "Unit1.Em4.ControlNodes".cmAnodeMainPnP1SuctionPlateVacuum.monitoring.error )
      Coil( "Unit1.Em4.ControlNodes".cmAnodeMainPnP1SuctionPlateVacuum.commands.reset )
   END_RUNG
   RUNG wire#w2
      Contact( "Unit1.Em4.ControlNodes".cmAnodeMainPnP2SuctionPlateVacuum.monitoring.error )
      Coil( "Unit1.Em4.ControlNodes".cmAnodeMainPnP2SuctionPlateVacuum.commands.reset )
   END_RUNG
   RUNG wire#w2
      Contact( "Unit1.Em4.ControlNodes".cmAnodeConveyorCoverFwdBwd.monitoring.error )
      Coil( "Unit1.Em4.ControlNodes".cmAnodeConveyorCoverFwdBwd.commands.reset )
   END_RUNG
   RUNG wire#w2
      Contact( "Unit1.Em4.ControlNodes".cmAnodeConveyorPickUpBlower.monitoring.error )
      Coil( "Unit1.Em4.ControlNodes".cmAnodeConveyorPickUpBlower.commands.reset )
   END_RUNG
   RUNG wire#w2
      Contact( "Unit1.Em4.ControlNodes".cmAnodeAlignTableSuctionPlateVacuum.monitoring.error )
      Coil( "Unit1.Em4.ControlNodes".cmAnodeAlignTableSuctionPlateVacuum.commands.reset )
   END_RUNG
   RUNG wire#w2
      Contact( "Unit1.Em4.ControlNodes".cmAnodeGlassCleaning.monitoring.error )
      Coil( "Unit1.Em4.ControlNodes".cmAnodeGlassCleaning.commands.reset )
   END_RUNG
   RUNG wire#powerrail
      Contact( #statUnitStatus.safetyReleased )
      wire#w3
      Contact( #statUnitStatus.acknowledgeActive )
      wire#w4
      Contact( "Unit1.Em4.ControlNodes".cmAnodeNgPnpUpDown.monitoring.error )
      Coil( "Unit1.Em4.ControlNodes".cmAnodeNgPnpUpDown.commands.reset )
   END_RUNG
   RUNG wire#w3
      Contact( #statUnitStatus.state.resetting )
   END_RUNG wire#w4
   RUNG wire#w4
      Contact( "Unit1.Em4.ControlNodes".cmAnodeNgPnp1stFwdBwd.monitoring.error )
      Coil( "Unit1.Em4.ControlNodes".cmAnodeNgPnp1stFwdBwd.commands.reset )
   END_RUNG
   RUNG wire#w4
      Contact( "Unit1.Em4.ControlNodes".cmAnodeNgPnp2ndFwdBwd.monitoring.error )
      Coil( "Unit1.Em4.ControlNodes".cmAnodeNgPnp2ndFwdBwd.commands.reset )
   END_RUNG
   RUNG wire#w4
      Contact( "Unit1.Em4.ControlNodes".cmAnodeNgPnpVaccum.monitoring.error )
      Coil( "Unit1.Em4.ControlNodes".cmAnodeNgPnpVaccum.commands.reset )
   END_RUNG
   RUNG wire#w4
      Contact( "Unit1.Em4.ControlNodes".cmAnodeMaintenanceMovingFixFwdBwd.monitoring.error )
      Coil( "Unit1.Em4.ControlNodes".cmAnodeMaintenanceMovingFixFwdBwd.commands.reset )
   END_RUNG
   RUNG wire#powerrail
      Contact( #statUnitStatus.safetyReleased )
      wire#w5
      Contact( #statUnitStatus.acknowledgeActive )
      wire#w6
      Contact( "Unit1.Em4.ControlNodes".cmAnodeNgBoxLiftUpDown.monitoring.error )
      Coil( "Unit1.Em4.ControlNodes".cmAnodeNgBoxLiftUpDown.commands.reset )
   END_RUNG
   RUNG wire#w5
      Contact( #statUnitStatus.state.resetting )
   END_RUNG wire#w6
   RUNG wire#w6
      Contact( "Unit1.Em4.ControlNodes".cmAnodeNgBoxLockUpDown.monitoring.error )
      Coil( "Unit1.Em4.ControlNodes".cmAnodeNgBoxLockUpDown.commands.reset )
   END_RUNG
   // the same network as SCL:
   #_w1 := #statUnitStatus.safetyReleased AND (#statUnitStatus.acknowledgeActive OR #statUnitStatus.state.resetting);
   "Unit1.Em4.ControlNodes".cmAnodeMainPnP1RotaryCwCcw.commands.reset := #_w1 AND "Unit1.Em4.ControlNodes".cmAnodeMainPnP1RotaryCwCcw.monitoring.error;
   "Unit1.Em4.ControlNodes".cmAnodeMainPnP1SuctionPlateVacuum.commands.reset := #_w1 AND "Unit1.Em4.ControlNodes".cmAnodeMainPnP1SuctionPlateVacuum.monitoring.error;
   "Unit1.Em4.ControlNodes".cmAnodeMainPnP2SuctionPlateVacuum.commands.reset := #_w1 AND "Unit1.Em4.ControlNodes".cmAnodeMainPnP2SuctionPlateVacuum.monitoring.error;
   "Unit1.Em4.ControlNodes".cmAnodeConveyorCoverFwdBwd.commands.reset := #_w1 AND "Unit1.Em4.ControlNodes".cmAnodeConveyorCoverFwdBwd.monitoring.error;
   "Unit1.Em4.ControlNodes".cmAnodeConveyorPickUpBlower.commands.reset := #_w1 AND "Unit1.Em4.ControlNodes".cmAnodeConveyorPickUpBlower.monitoring.error;
   "Unit1.Em4.ControlNodes".cmAnodeAlignTableSuctionPlateVacuum.commands.reset := #_w1 AND "Unit1.Em4.ControlNodes".cmAnodeAlignTableSuctionPlateVacuum.monitoring.error;
   "Unit1.Em4.ControlNodes".cmAnodeGlassCleaning.commands.reset := #_w1 AND "Unit1.Em4.ControlNodes".cmAnodeGlassCleaning.monitoring.error;
   #_w2 := #statUnitStatus.safetyReleased AND (#statUnitStatus.acknowledgeActive OR #statUnitStatus.state.resetting);
   "Unit1.Em4.ControlNodes".cmAnodeNgPnpUpDown.commands.reset := #_w2 AND "Unit1.Em4.ControlNodes".cmAnodeNgPnpUpDown.monitoring.error;
   "Unit1.Em4.ControlNodes".cmAnodeNgPnp1stFwdBwd.commands.reset := #_w2 AND "Unit1.Em4.ControlNodes".cmAnodeNgPnp1stFwdBwd.monitoring.error;
   "Unit1.Em4.ControlNodes".cmAnodeNgPnp2ndFwdBwd.commands.reset := #_w2 AND "Unit1.Em4.ControlNodes".cmAnodeNgPnp2ndFwdBwd.monitoring.error;
   "Unit1.Em4.ControlNodes".cmAnodeNgPnpVaccum.commands.reset := #_w2 AND "Unit1.Em4.ControlNodes".cmAnodeNgPnpVaccum.monitoring.error;
   "Unit1.Em4.ControlNodes".cmAnodeMaintenanceMovingFixFwdBwd.commands.reset := #_w2 AND "Unit1.Em4.ControlNodes".cmAnodeMaintenanceMovingFixFwdBwd.monitoring.error;
   #_w3 := #statUnitStatus.safetyReleased AND (#statUnitStatus.acknowledgeActive OR #statUnitStatus.state.resetting);
   "Unit1.Em4.ControlNodes".cmAnodeNgBoxLiftUpDown.commands.reset := #_w3 AND "Unit1.Em4.ControlNodes".cmAnodeNgBoxLiftUpDown.monitoring.error;
   "Unit1.Em4.ControlNodes".cmAnodeNgBoxLockUpDown.commands.reset := #_w3 AND "Unit1.Em4.ControlNodes".cmAnodeNgBoxLockUpDown.monitoring.error;
END_REGION

REGION Network 227: CmAnodeMainPnP1RotaryCwCcw Home
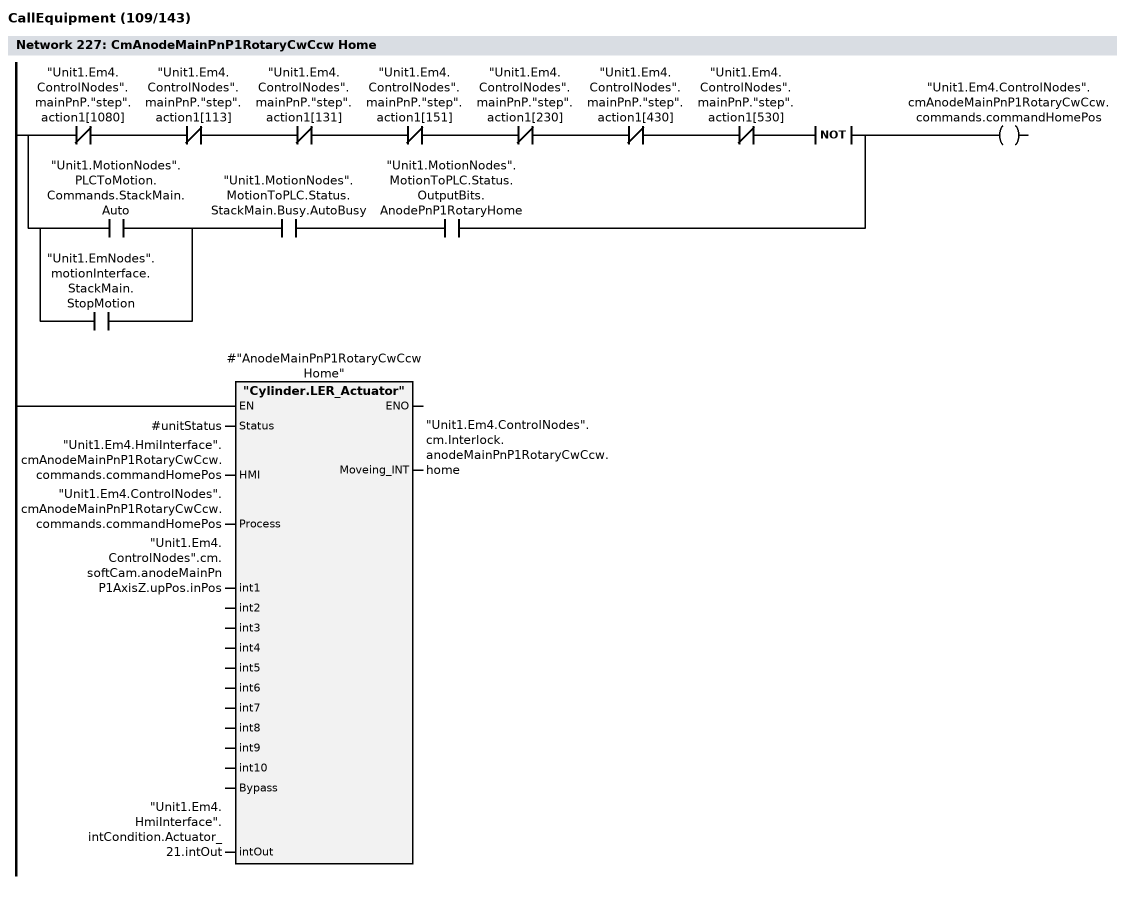
   RUNG wire#powerrail
      I_Contact( "Unit1.Em4.ControlNodes".mainPnP."step".action1[1080] )
      I_Contact( "Unit1.Em4.ControlNodes".mainPnP."step".action1[113] )
      I_Contact( "Unit1.Em4.ControlNodes".mainPnP."step".action1[131] )
      I_Contact( "Unit1.Em4.ControlNodes".mainPnP."step".action1[151] )
      I_Contact( "Unit1.Em4.ControlNodes".mainPnP."step".action1[230] )
      I_Contact( "Unit1.Em4.ControlNodes".mainPnP."step".action1[430] )
      I_Contact( "Unit1.Em4.ControlNodes".mainPnP."step".action1[530] )
      Not()
      wire#w1
      Coil( "Unit1.Em4.ControlNodes".cmAnodeMainPnP1RotaryCwCcw.commands.commandHomePos )
   END_RUNG
   RUNG wire#powerrail
      Contact( "Unit1.MotionNodes".PLCToMotion.Commands.StackMain.Auto )
      wire#w2
      Contact( "Unit1.MotionNodes".MotionToPLC.Status.StackMain.Busy.AutoBusy )
      Contact( "Unit1.MotionNodes".MotionToPLC.Status.OutputBits.AnodePnP1RotaryHome )
   END_RUNG wire#w1
   RUNG wire#powerrail
      Contact( "Unit1.EmNodes".motionInterface.StackMain.StopMotion )
   END_RUNG wire#w2
   RUNG wire#powerrail
      #"AnodeMainPnP1RotaryCwCcw Home"(Status := #unitStatus, HMI := "Unit1.Em4.HmiInterface".cmAnodeMainPnP1RotaryCwCcw.commands.commandHomePos, Process := "Unit1.Em4.ControlNodes".cmAnodeMainPnP1RotaryCwCcw.commands.commandHomePos, int1 := "Unit1.Em4.ControlNodes".cm.softCam.anodeMainPnP1AxisZ.upPos.inPos, int2 :=, int3 :=, int4 :=, int5 :=, int6 :=, int7 :=, int8 :=, int9 :=, int10 :=, Bypass :=, intOut := "Unit1.Em4.HmiInterface".intCondition.Actuator_21.intOut, Moveing_INT => "Unit1.Em4.ControlNodes".cm.Interlock.anodeMainPnP1RotaryCwCcw.home)
   END_RUNG
   // the same network as SCL:
   "Unit1.Em4.ControlNodes".cmAnodeMainPnP1RotaryCwCcw.commands.commandHomePos := NOT (NOT "Unit1.Em4.ControlNodes".mainPnP."step".action1[1080] AND NOT "Unit1.Em4.ControlNodes".mainPnP."step".action1[113] AND NOT "Unit1.Em4.ControlNodes".mainPnP."step".action1[131] AND NOT "Unit1.Em4.ControlNodes".mainPnP."step".action1[151] AND NOT "Unit1.Em4.ControlNodes".mainPnP."step".action1[230] AND NOT "Unit1.Em4.ControlNodes".mainPnP."step".action1[430] AND NOT "Unit1.Em4.ControlNodes".mainPnP."step".action1[530]) OR (("Unit1.MotionNodes".PLCToMotion.Commands.StackMain.Auto OR "Unit1.EmNodes".motionInterface.StackMain.StopMotion) AND "Unit1.MotionNodes".MotionToPLC.Status.StackMain.Busy.AutoBusy AND "Unit1.MotionNodes".MotionToPLC.Status.OutputBits.AnodePnP1RotaryHome);
   #"AnodeMainPnP1RotaryCwCcw Home"(Status := #unitStatus,   // "Cylinder.LER_Actuator"
                           HMI := "Unit1.Em4.HmiInterface".cmAnodeMainPnP1RotaryCwCcw.commands.commandHomePos,
                           Process := "Unit1.Em4.ControlNodes".cmAnodeMainPnP1RotaryCwCcw.commands.commandHomePos,
                           int1 := "Unit1.Em4.ControlNodes".cm.softCam.anodeMainPnP1AxisZ.upPos.inPos,
                           intOut := "Unit1.Em4.HmiInterface".intCondition.Actuator_21.intOut,
                           Moveing_INT => "Unit1.Em4.ControlNodes".cm.Interlock.anodeMainPnP1RotaryCwCcw.home);
END_REGION

REGION Network 228: CmAnodeMainPnP1RotaryCwCcw Work
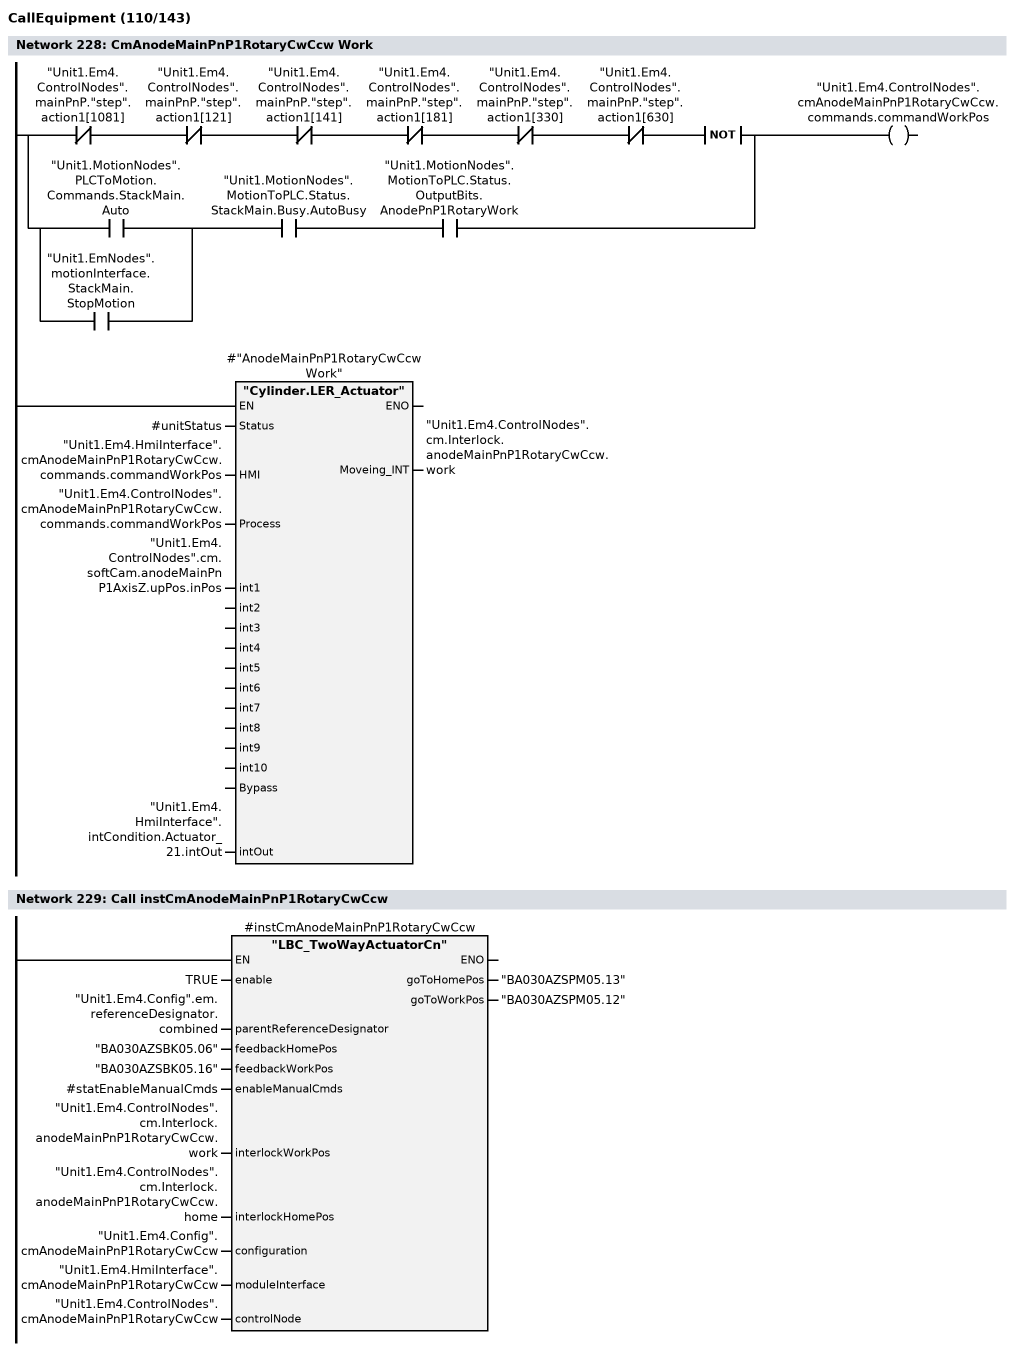
   RUNG wire#powerrail
      I_Contact( "Unit1.Em4.ControlNodes".mainPnP."step".action1[1081] )
      I_Contact( "Unit1.Em4.ControlNodes".mainPnP."step".action1[121] )
      I_Contact( "Unit1.Em4.ControlNodes".mainPnP."step".action1[141] )
      I_Contact( "Unit1.Em4.ControlNodes".mainPnP."step".action1[181] )
      I_Contact( "Unit1.Em4.ControlNodes".mainPnP."step".action1[330] )
      I_Contact( "Unit1.Em4.ControlNodes".mainPnP."step".action1[630] )
      Not()
      wire#w1
      Coil( "Unit1.Em4.ControlNodes".cmAnodeMainPnP1RotaryCwCcw.commands.commandWorkPos )
   END_RUNG
   RUNG wire#powerrail
      Contact( "Unit1.MotionNodes".PLCToMotion.Commands.StackMain.Auto )
      wire#w2
      Contact( "Unit1.MotionNodes".MotionToPLC.Status.StackMain.Busy.AutoBusy )
      Contact( "Unit1.MotionNodes".MotionToPLC.Status.OutputBits.AnodePnP1RotaryWork )
   END_RUNG wire#w1
   RUNG wire#powerrail
      Contact( "Unit1.EmNodes".motionInterface.StackMain.StopMotion )
   END_RUNG wire#w2
   RUNG wire#powerrail
      #"AnodeMainPnP1RotaryCwCcw Work"(Status := #unitStatus, HMI := "Unit1.Em4.HmiInterface".cmAnodeMainPnP1RotaryCwCcw.commands.commandWorkPos, Process := "Unit1.Em4.ControlNodes".cmAnodeMainPnP1RotaryCwCcw.commands.commandWorkPos, int1 := "Unit1.Em4.ControlNodes".cm.softCam.anodeMainPnP1AxisZ.upPos.inPos, int2 :=, int3 :=, int4 :=, int5 :=, int6 :=, int7 :=, int8 :=, int9 :=, int10 :=, Bypass :=, intOut := "Unit1.Em4.HmiInterface".intCondition.Actuator_21.intOut, Moveing_INT => "Unit1.Em4.ControlNodes".cm.Interlock.anodeMainPnP1RotaryCwCcw.work)
   END_RUNG
   // the same network as SCL:
   "Unit1.Em4.ControlNodes".cmAnodeMainPnP1RotaryCwCcw.commands.commandWorkPos := NOT (NOT "Unit1.Em4.ControlNodes".mainPnP."step".action1[1081] AND NOT "Unit1.Em4.ControlNodes".mainPnP."step".action1[121] AND NOT "Unit1.Em4.ControlNodes".mainPnP."step".action1[141] AND NOT "Unit1.Em4.ControlNodes".mainPnP."step".action1[181] AND NOT "Unit1.Em4.ControlNodes".mainPnP."step".action1[330] AND NOT "Unit1.Em4.ControlNodes".mainPnP."step".action1[630]) OR (("Unit1.MotionNodes".PLCToMotion.Commands.StackMain.Auto OR "Unit1.EmNodes".motionInterface.StackMain.StopMotion) AND "Unit1.MotionNodes".MotionToPLC.Status.StackMain.Busy.AutoBusy AND "Unit1.MotionNodes".MotionToPLC.Status.OutputBits.AnodePnP1RotaryWork);
   #"AnodeMainPnP1RotaryCwCcw Work"(Status := #unitStatus,   // "Cylinder.LER_Actuator"
                           HMI := "Unit1.Em4.HmiInterface".cmAnodeMainPnP1RotaryCwCcw.commands.commandWorkPos,
                           Process := "Unit1.Em4.ControlNodes".cmAnodeMainPnP1RotaryCwCcw.commands.commandWorkPos,
                           int1 := "Unit1.Em4.ControlNodes".cm.softCam.anodeMainPnP1AxisZ.upPos.inPos,
                           intOut := "Unit1.Em4.HmiInterface".intCondition.Actuator_21.intOut,
                           Moveing_INT => "Unit1.Em4.ControlNodes".cm.Interlock.anodeMainPnP1RotaryCwCcw.work);
END_REGION

REGION Network 229: Call instCmAnodeMainPnP1RotaryCwCcw
   RUNG wire#powerrail
      #instCmAnodeMainPnP1RotaryCwCcw(enable := TRUE, parentReferenceDesignator := "Unit1.Em4.Config".em.referenceDesignator.combined, feedbackHomePos := "BA030AZSBK05.06", feedbackWorkPos := "BA030AZSBK05.16", enableManualCmds := #statEnableManualCmds, interlockWorkPos := "Unit1.Em4.ControlNodes".cm.Interlock.anodeMainPnP1RotaryCwCcw.work, interlockHomePos := "Unit1.Em4.ControlNodes".cm.Interlock.anodeMainPnP1RotaryCwCcw.home, configuration := "Unit1.Em4.Config".cmAnodeMainPnP1RotaryCwCcw, moduleInterface := "Unit1.Em4.HmiInterface".cmAnodeMainPnP1RotaryCwCcw, controlNode := "Unit1.Em4.ControlNodes".cmAnodeMainPnP1RotaryCwCcw, goToHomePos => "BA030AZSPM05.13", goToWorkPos => "BA030AZSPM05.12")
   END_RUNG
   // the same network as SCL:
   #instCmAnodeMainPnP1RotaryCwCcw(enable := TRUE,   // "LBC_TwoWayActuatorCn"
                           parentReferenceDesignator := "Unit1.Em4.Config".em.referenceDesignator.combined,
                           feedbackHomePos := "BA030AZSBK05.06",
                           feedbackWorkPos := "BA030AZSBK05.16",
                           enableManualCmds := #statEnableManualCmds,
                           interlockWorkPos := "Unit1.Em4.ControlNodes".cm.Interlock.anodeMainPnP1RotaryCwCcw.work,
                           interlockHomePos := "Unit1.Em4.ControlNodes".cm.Interlock.anodeMainPnP1RotaryCwCcw.home,
                           configuration := "Unit1.Em4.Config".cmAnodeMainPnP1RotaryCwCcw,
                           moduleInterface := "Unit1.Em4.HmiInterface".cmAnodeMainPnP1RotaryCwCcw,
                           controlNode := "Unit1.Em4.ControlNodes".cmAnodeMainPnP1RotaryCwCcw,
                           goToHomePos => "BA030AZSPM05.13",
                           goToWorkPos => "BA030AZSPM05.12");
END_REGION

REGION Network 231: CmAnodeMainPnP1SuctionPlateVacuum Home
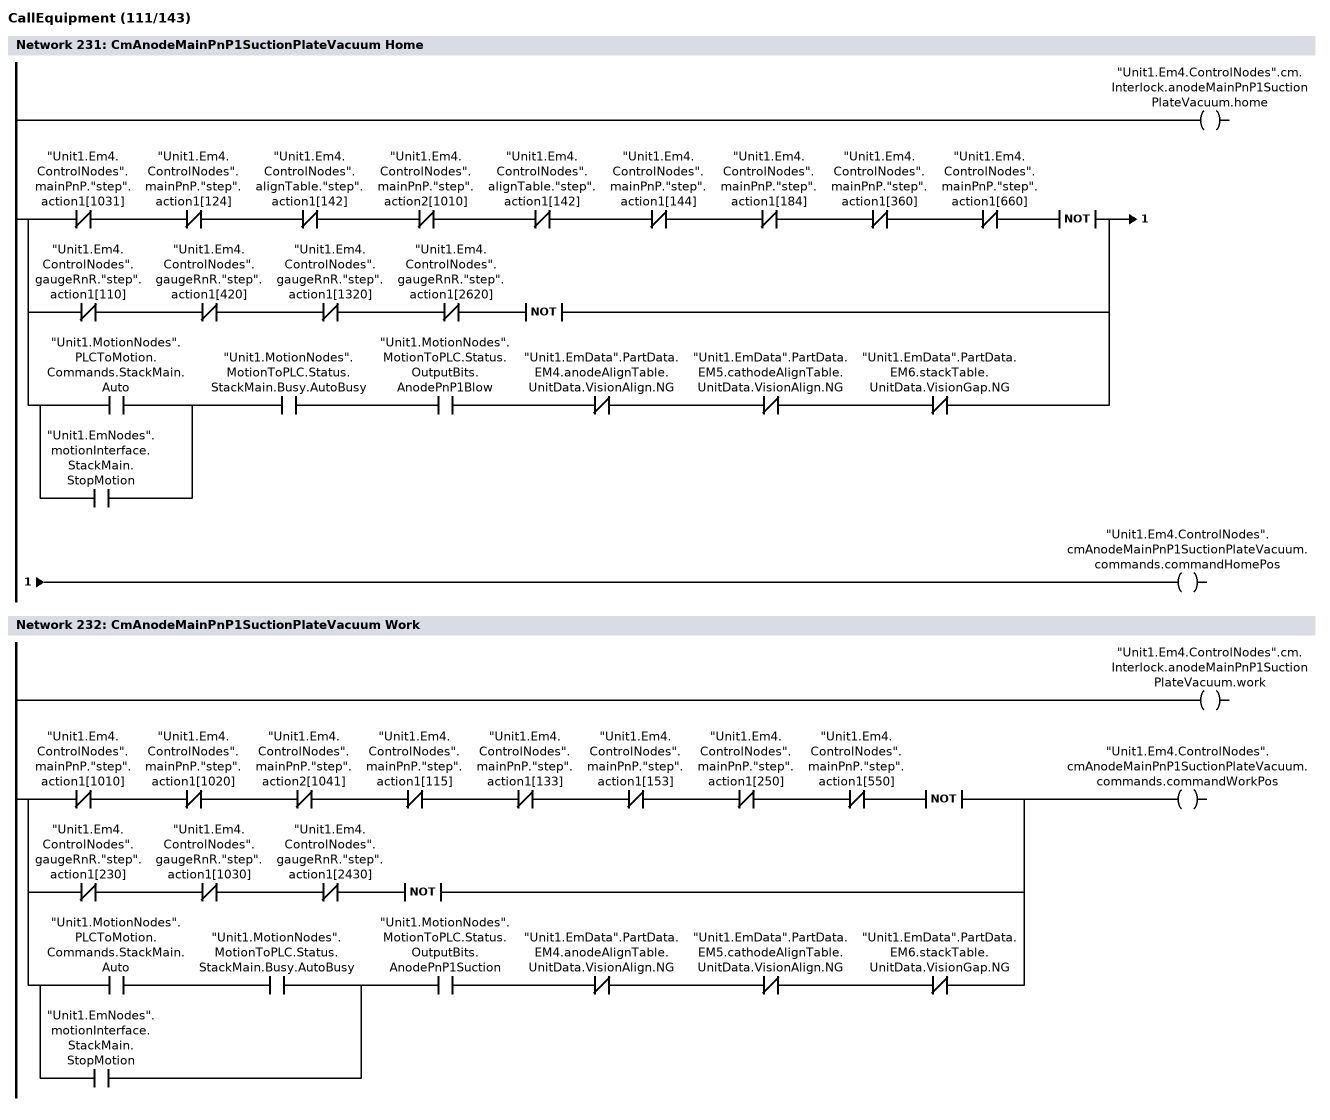
   RUNG wire#powerrail
      Coil( "Unit1.Em4.ControlNodes".cm.Interlock.anodeMainPnP1SuctionPlateVacuum.home )
   END_RUNG
   RUNG wire#powerrail
      I_Contact( "Unit1.Em4.ControlNodes".mainPnP."step".action1[1031] )
      I_Contact( "Unit1.Em4.ControlNodes".mainPnP."step".action1[124] )
      I_Contact( "Unit1.Em4.ControlNodes".alignTable."step".action1[142] )
      I_Contact( "Unit1.Em4.ControlNodes".mainPnP."step".action2[1010] )
      I_Contact( "Unit1.Em4.ControlNodes".alignTable."step".action1[142] )
      I_Contact( "Unit1.Em4.ControlNodes".mainPnP."step".action1[144] )
      I_Contact( "Unit1.Em4.ControlNodes".mainPnP."step".action1[184] )
      I_Contact( "Unit1.Em4.ControlNodes".mainPnP."step".action1[360] )
      I_Contact( "Unit1.Em4.ControlNodes".mainPnP."step".action1[660] )
      Not()
      wire#w1
      Coil( "Unit1.Em4.ControlNodes".cmAnodeMainPnP1SuctionPlateVacuum.commands.commandHomePos )
   END_RUNG
   RUNG wire#powerrail
      I_Contact( "Unit1.Em4.ControlNodes".gaugeRnR."step".action1[110] )
      I_Contact( "Unit1.Em4.ControlNodes".gaugeRnR."step".action1[420] )
      I_Contact( "Unit1.Em4.ControlNodes".gaugeRnR."step".action1[1320] )
      I_Contact( "Unit1.Em4.ControlNodes".gaugeRnR."step".action1[2620] )
      Not()
   END_RUNG wire#w1
   RUNG wire#powerrail
      Contact( "Unit1.MotionNodes".PLCToMotion.Commands.StackMain.Auto )
      wire#w2
      Contact( "Unit1.MotionNodes".MotionToPLC.Status.StackMain.Busy.AutoBusy )
      Contact( "Unit1.MotionNodes".MotionToPLC.Status.OutputBits.AnodePnP1Blow )
      I_Contact( "Unit1.EmData".PartData.EM4.anodeAlignTable.UnitData.VisionAlign.NG )
      I_Contact( "Unit1.EmData".PartData.EM5.cathodeAlignTable.UnitData.VisionAlign.NG )
      I_Contact( "Unit1.EmData".PartData.EM6.stackTable.UnitData.VisionGap.NG )
   END_RUNG wire#w1
   RUNG wire#powerrail
      Contact( "Unit1.EmNodes".motionInterface.StackMain.StopMotion )
   END_RUNG wire#w2
   // the same network as SCL:
   "Unit1.Em4.ControlNodes".cm.Interlock.anodeMainPnP1SuctionPlateVacuum.home := TRUE;
   "Unit1.Em4.ControlNodes".cmAnodeMainPnP1SuctionPlateVacuum.commands.commandHomePos := NOT (NOT "Unit1.Em4.ControlNodes".mainPnP."step".action1[1031] AND NOT "Unit1.Em4.ControlNodes".mainPnP."step".action1[124] AND NOT "Unit1.Em4.ControlNodes".alignTable."step".action1[142] AND NOT "Unit1.Em4.ControlNodes".mainPnP."step".action2[1010] AND NOT "Unit1.Em4.ControlNodes".alignTable."step".action1[142] AND NOT "Unit1.Em4.ControlNodes".mainPnP."step".action1[144] AND NOT "Unit1.Em4.ControlNodes".mainPnP."step".action1[184] AND NOT "Unit1.Em4.ControlNodes".mainPnP."step".action1[360] AND NOT "Unit1.Em4.ControlNodes".mainPnP."step".action1[660]) OR NOT (NOT "Unit1.Em4.ControlNodes".gaugeRnR."step".action1[110] AND NOT "Unit1.Em4.ControlNodes".gaugeRnR."step".action1[420] AND NOT "Unit1.Em4.ControlNodes".gaugeRnR."step".action1[1320] AND NOT "Unit1.Em4.ControlNodes".gaugeRnR."step".action1[2620]) OR (("Unit1.MotionNodes".PLCToMotion.Commands.StackMain.Auto OR "Unit1.EmNodes".motionInterface.StackMain.StopMotion) AND "Unit1.MotionNodes".MotionToPLC.Status.StackMain.Busy.AutoBusy AND "Unit1.MotionNodes".MotionToPLC.Status.OutputBits.AnodePnP1Blow AND NOT "Unit1.EmData".PartData.EM4.anodeAlignTable.UnitData.VisionAlign.NG AND NOT "Unit1.EmData".PartData.EM5.cathodeAlignTable.UnitData.VisionAlign.NG AND NOT "Unit1.EmData".PartData.EM6.stackTable.UnitData.VisionGap.NG);
END_REGION

REGION Network 232: CmAnodeMainPnP1SuctionPlateVacuum Work
   RUNG wire#powerrail
      Coil( "Unit1.Em4.ControlNodes".cm.Interlock.anodeMainPnP1SuctionPlateVacuum.work )
   END_RUNG
   RUNG wire#powerrail
      I_Contact( "Unit1.Em4.ControlNodes".mainPnP."step".action1[1010] )
      I_Contact( "Unit1.Em4.ControlNodes".mainPnP."step".action1[1020] )
      I_Contact( "Unit1.Em4.ControlNodes".mainPnP."step".action2[1041] )
      I_Contact( "Unit1.Em4.ControlNodes".mainPnP."step".action1[115] )
      I_Contact( "Unit1.Em4.ControlNodes".mainPnP."step".action1[133] )
      I_Contact( "Unit1.Em4.ControlNodes".mainPnP."step".action1[153] )
      I_Contact( "Unit1.Em4.ControlNodes".mainPnP."step".action1[250] )
      I_Contact( "Unit1.Em4.ControlNodes".mainPnP."step".action1[550] )
      Not()
      wire#w1
      Coil( "Unit1.Em4.ControlNodes".cmAnodeMainPnP1SuctionPlateVacuum.commands.commandWorkPos )
   END_RUNG
   RUNG wire#powerrail
      I_Contact( "Unit1.Em4.ControlNodes".gaugeRnR."step".action1[230] )
      I_Contact( "Unit1.Em4.ControlNodes".gaugeRnR."step".action1[1030] )
      I_Contact( "Unit1.Em4.ControlNodes".gaugeRnR."step".action1[2430] )
      Not()
   END_RUNG wire#w1
   RUNG wire#powerrail
      Contact( "Unit1.MotionNodes".PLCToMotion.Commands.StackMain.Auto )
      Contact( "Unit1.MotionNodes".MotionToPLC.Status.StackMain.Busy.AutoBusy )
      wire#w2
      Contact( "Unit1.MotionNodes".MotionToPLC.Status.OutputBits.AnodePnP1Suction )
      I_Contact( "Unit1.EmData".PartData.EM4.anodeAlignTable.UnitData.VisionAlign.NG )
      I_Contact( "Unit1.EmData".PartData.EM5.cathodeAlignTable.UnitData.VisionAlign.NG )
      I_Contact( "Unit1.EmData".PartData.EM6.stackTable.UnitData.VisionGap.NG )
   END_RUNG wire#w1
   RUNG wire#powerrail
      Contact( "Unit1.EmNodes".motionInterface.StackMain.StopMotion )
   END_RUNG wire#w2
   // the same network as SCL:
   "Unit1.Em4.ControlNodes".cm.Interlock.anodeMainPnP1SuctionPlateVacuum.work := TRUE;
   "Unit1.Em4.ControlNodes".cmAnodeMainPnP1SuctionPlateVacuum.commands.commandWorkPos := NOT (NOT "Unit1.Em4.ControlNodes".mainPnP."step".action1[1010] AND NOT "Unit1.Em4.ControlNodes".mainPnP."step".action1[1020] AND NOT "Unit1.Em4.ControlNodes".mainPnP."step".action2[1041] AND NOT "Unit1.Em4.ControlNodes".mainPnP."step".action1[115] AND NOT "Unit1.Em4.ControlNodes".mainPnP."step".action1[133] AND NOT "Unit1.Em4.ControlNodes".mainPnP."step".action1[153] AND NOT "Unit1.Em4.ControlNodes".mainPnP."step".action1[250] AND NOT "Unit1.Em4.ControlNodes".mainPnP."step".action1[550]) OR NOT (NOT "Unit1.Em4.ControlNodes".gaugeRnR."step".action1[230] AND NOT "Unit1.Em4.ControlNodes".gaugeRnR."step".action1[1030] AND NOT "Unit1.Em4.ControlNodes".gaugeRnR."step".action1[2430]) OR ((("Unit1.MotionNodes".PLCToMotion.Commands.StackMain.Auto AND "Unit1.MotionNodes".MotionToPLC.Status.StackMain.Busy.AutoBusy) OR "Unit1.EmNodes".motionInterface.StackMain.StopMotion) AND "Unit1.MotionNodes".MotionToPLC.Status.OutputBits.AnodePnP1Suction AND NOT "Unit1.EmData".PartData.EM4.anodeAlignTable.UnitData.VisionAlign.NG AND NOT "Unit1.EmData".PartData.EM5.cathodeAlignTable.UnitData.VisionAlign.NG AND NOT "Unit1.EmData".PartData.EM6.stackTable.UnitData.VisionGap.NG);
END_REGION

REGION Network 233: Call instCmAnodeMainPnP1SuctionPlateVacuum
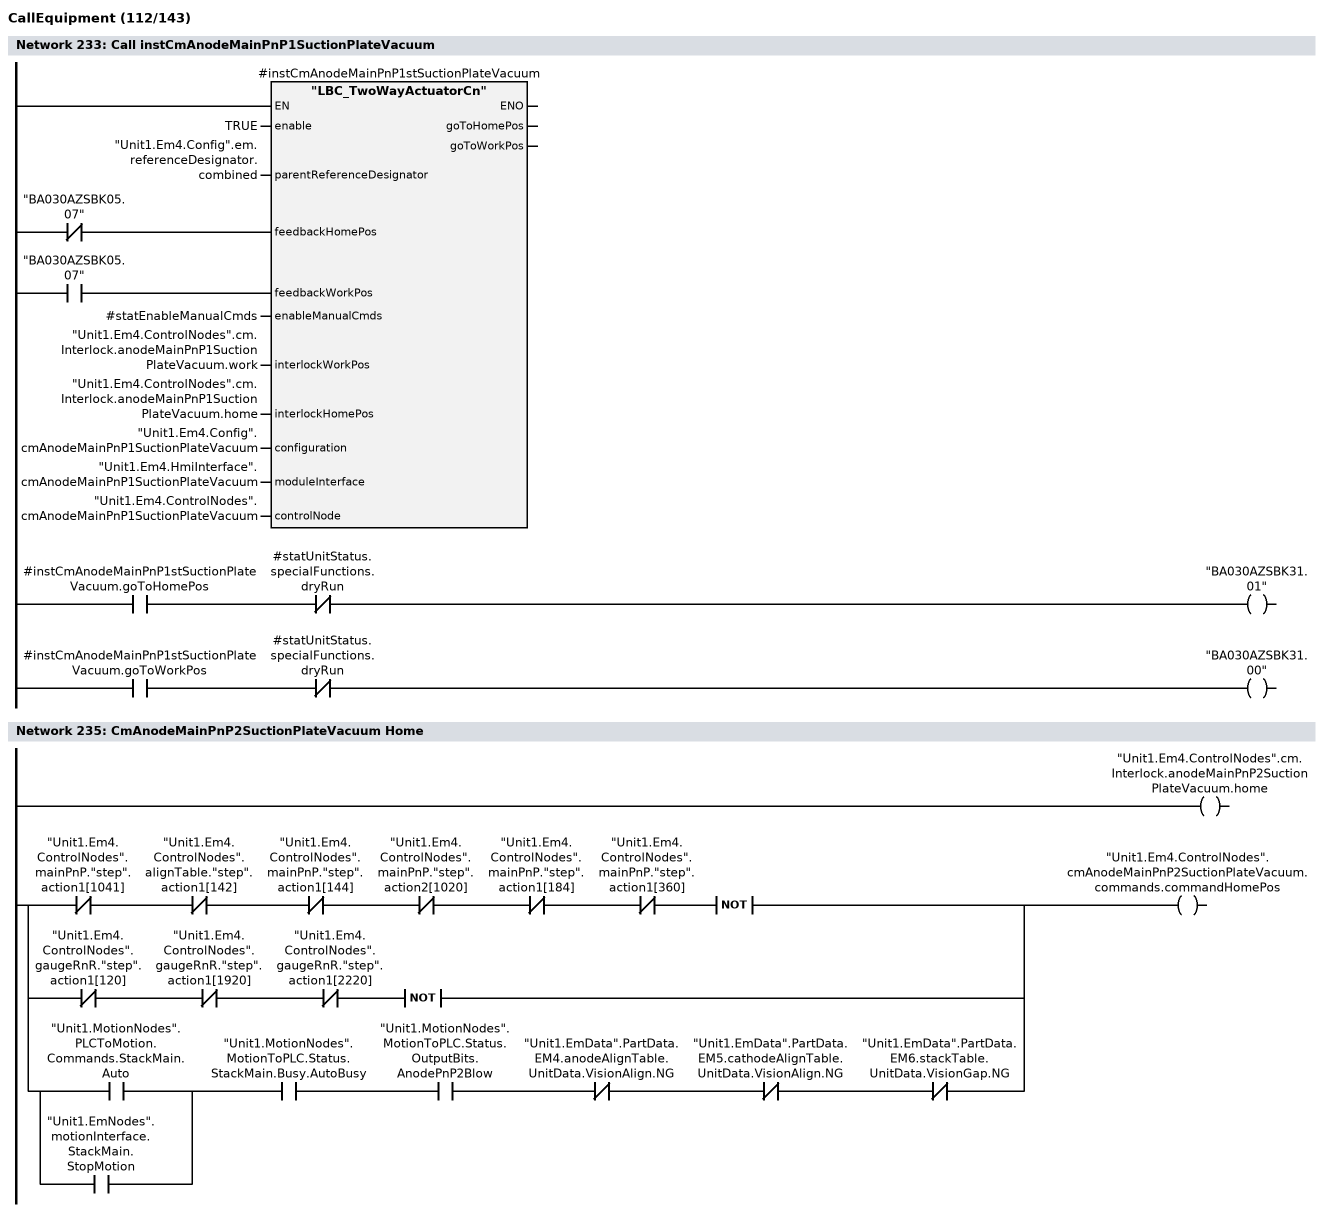
   RUNG wire#powerrail
      #instCmAnodeMainPnP1stSuctionPlateVacuum(feedbackHomePos := wire#w1, feedbackWorkPos := wire#w2, enable := TRUE, parentReferenceDesignator := "Unit1.Em4.Config".em.referenceDesignator.combined, enableManualCmds := #statEnableManualCmds, interlockWorkPos := "Unit1.Em4.ControlNodes".cm.Interlock.anodeMainPnP1SuctionPlateVacuum.work, interlockHomePos := "Unit1.Em4.ControlNodes".cm.Interlock.anodeMainPnP1SuctionPlateVacuum.home, configuration := "Unit1.Em4.Config".cmAnodeMainPnP1SuctionPlateVacuum, moduleInterface := "Unit1.Em4.HmiInterface".cmAnodeMainPnP1SuctionPlateVacuum, controlNode := "Unit1.Em4.ControlNodes".cmAnodeMainPnP1SuctionPlateVacuum, goToHomePos =>, goToWorkPos =>)
   END_RUNG
   RUNG wire#powerrail
      I_Contact( "BA030AZSBK05.07" )
   END_RUNG wire#w1
   RUNG wire#powerrail
      Contact( "BA030AZSBK05.07" )
   END_RUNG wire#w2
   RUNG wire#powerrail
      Contact( #instCmAnodeMainPnP1stSuctionPlateVacuum.goToHomePos )
      I_Contact( #statUnitStatus.specialFunctions.dryRun )
      Coil( "BA030AZSBK31.01" )
   END_RUNG
   RUNG wire#powerrail
      Contact( #instCmAnodeMainPnP1stSuctionPlateVacuum.goToWorkPos )
      I_Contact( #statUnitStatus.specialFunctions.dryRun )
      Coil( "BA030AZSBK31.00" )
   END_RUNG
   // the same network as SCL:
   #instCmAnodeMainPnP1stSuctionPlateVacuum(enable := TRUE,   // "LBC_TwoWayActuatorCn"
                           parentReferenceDesignator := "Unit1.Em4.Config".em.referenceDesignator.combined,
                           feedbackHomePos := NOT "BA030AZSBK05.07",
                           feedbackWorkPos := "BA030AZSBK05.07",
                           enableManualCmds := #statEnableManualCmds,
                           interlockWorkPos := "Unit1.Em4.ControlNodes".cm.Interlock.anodeMainPnP1SuctionPlateVacuum.work,
                           interlockHomePos := "Unit1.Em4.ControlNodes".cm.Interlock.anodeMainPnP1SuctionPlateVacuum.home,
                           configuration := "Unit1.Em4.Config".cmAnodeMainPnP1SuctionPlateVacuum,
                           moduleInterface := "Unit1.Em4.HmiInterface".cmAnodeMainPnP1SuctionPlateVacuum,
                           controlNode := "Unit1.Em4.ControlNodes".cmAnodeMainPnP1SuctionPlateVacuum);
   "BA030AZSBK31.01" := #instCmAnodeMainPnP1stSuctionPlateVacuum.goToHomePos AND NOT #statUnitStatus.specialFunctions.dryRun;
   "BA030AZSBK31.00" := #instCmAnodeMainPnP1stSuctionPlateVacuum.goToWorkPos AND NOT #statUnitStatus.specialFunctions.dryRun;
END_REGION

REGION Network 235: CmAnodeMainPnP2SuctionPlateVacuum Home
   RUNG wire#powerrail
      Coil( "Unit1.Em4.ControlNodes".cm.Interlock.anodeMainPnP2SuctionPlateVacuum.home )
   END_RUNG
   RUNG wire#powerrail
      I_Contact( "Unit1.Em4.ControlNodes".mainPnP."step".action1[1041] )
      I_Contact( "Unit1.Em4.ControlNodes".alignTable."step".action1[142] )
      I_Contact( "Unit1.Em4.ControlNodes".mainPnP."step".action1[144] )
      I_Contact( "Unit1.Em4.ControlNodes".mainPnP."step".action2[1020] )
      I_Contact( "Unit1.Em4.ControlNodes".mainPnP."step".action1[184] )
      I_Contact( "Unit1.Em4.ControlNodes".mainPnP."step".action1[360] )
      Not()
      wire#w1
      Coil( "Unit1.Em4.ControlNodes".cmAnodeMainPnP2SuctionPlateVacuum.commands.commandHomePos )
   END_RUNG
   RUNG wire#powerrail
      I_Contact( "Unit1.Em4.ControlNodes".gaugeRnR."step".action1[120] )
      I_Contact( "Unit1.Em4.ControlNodes".gaugeRnR."step".action1[1920] )
      I_Contact( "Unit1.Em4.ControlNodes".gaugeRnR."step".action1[2220] )
      Not()
   END_RUNG wire#w1
   RUNG wire#powerrail
      Contact( "Unit1.MotionNodes".PLCToMotion.Commands.StackMain.Auto )
      wire#w2
      Contact( "Unit1.MotionNodes".MotionToPLC.Status.StackMain.Busy.AutoBusy )
      Contact( "Unit1.MotionNodes".MotionToPLC.Status.OutputBits.AnodePnP2Blow )
      I_Contact( "Unit1.EmData".PartData.EM4.anodeAlignTable.UnitData.VisionAlign.NG )
      I_Contact( "Unit1.EmData".PartData.EM5.cathodeAlignTable.UnitData.VisionAlign.NG )
      I_Contact( "Unit1.EmData".PartData.EM6.stackTable.UnitData.VisionGap.NG )
   END_RUNG wire#w1
   RUNG wire#powerrail
      Contact( "Unit1.EmNodes".motionInterface.StackMain.StopMotion )
   END_RUNG wire#w2
   // the same network as SCL:
   "Unit1.Em4.ControlNodes".cm.Interlock.anodeMainPnP2SuctionPlateVacuum.home := TRUE;
   "Unit1.Em4.ControlNodes".cmAnodeMainPnP2SuctionPlateVacuum.commands.commandHomePos := NOT (NOT "Unit1.Em4.ControlNodes".mainPnP."step".action1[1041] AND NOT "Unit1.Em4.ControlNodes".alignTable."step".action1[142] AND NOT "Unit1.Em4.ControlNodes".mainPnP."step".action1[144] AND NOT "Unit1.Em4.ControlNodes".mainPnP."step".action2[1020] AND NOT "Unit1.Em4.ControlNodes".mainPnP."step".action1[184] AND NOT "Unit1.Em4.ControlNodes".mainPnP."step".action1[360]) OR NOT (NOT "Unit1.Em4.ControlNodes".gaugeRnR."step".action1[120] AND NOT "Unit1.Em4.ControlNodes".gaugeRnR."step".action1[1920] AND NOT "Unit1.Em4.ControlNodes".gaugeRnR."step".action1[2220]) OR (("Unit1.MotionNodes".PLCToMotion.Commands.StackMain.Auto OR "Unit1.EmNodes".motionInterface.StackMain.StopMotion) AND "Unit1.MotionNodes".MotionToPLC.Status.StackMain.Busy.AutoBusy AND "Unit1.MotionNodes".MotionToPLC.Status.OutputBits.AnodePnP2Blow AND NOT "Unit1.EmData".PartData.EM4.anodeAlignTable.UnitData.VisionAlign.NG AND NOT "Unit1.EmData".PartData.EM5.cathodeAlignTable.UnitData.VisionAlign.NG AND NOT "Unit1.EmData".PartData.EM6.stackTable.UnitData.VisionGap.NG);
END_REGION

REGION Network 236: CmAnodeMainPnP2SuctionPlateVacuum Work
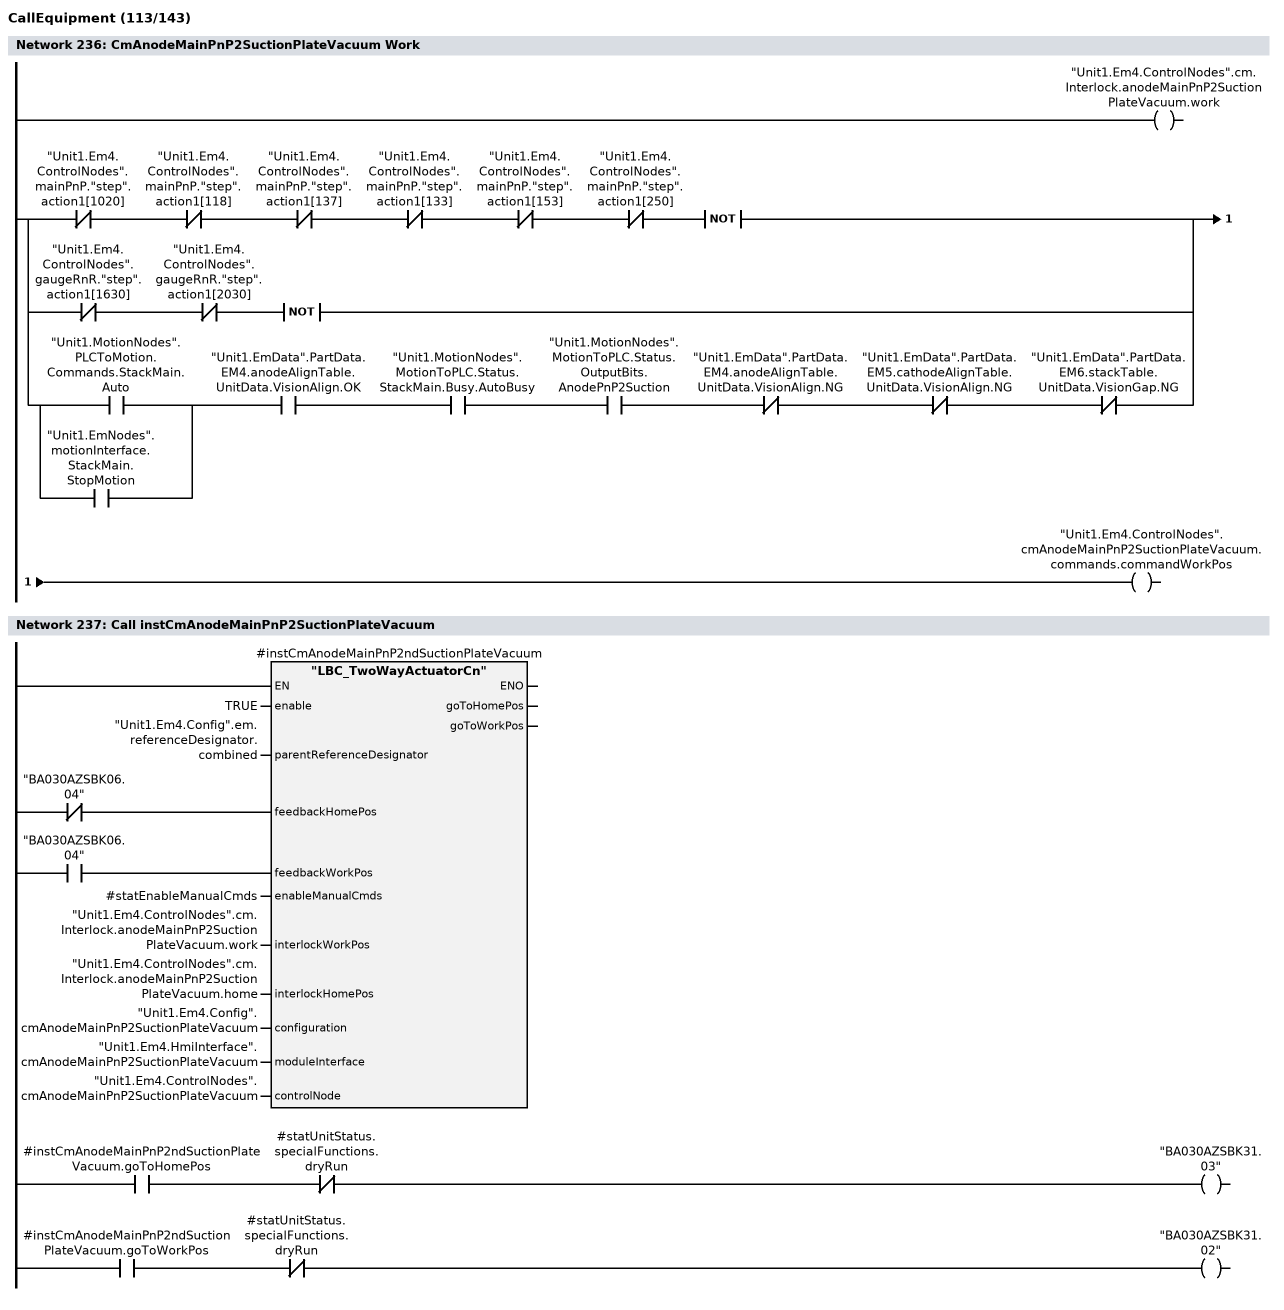
   RUNG wire#powerrail
      Coil( "Unit1.Em4.ControlNodes".cm.Interlock.anodeMainPnP2SuctionPlateVacuum.work )
   END_RUNG
   RUNG wire#powerrail
      I_Contact( "Unit1.Em4.ControlNodes".mainPnP."step".action1[1020] )
      I_Contact( "Unit1.Em4.ControlNodes".mainPnP."step".action1[118] )
      I_Contact( "Unit1.Em4.ControlNodes".mainPnP."step".action1[137] )
      I_Contact( "Unit1.Em4.ControlNodes".mainPnP."step".action1[133] )
      I_Contact( "Unit1.Em4.ControlNodes".mainPnP."step".action1[153] )
      I_Contact( "Unit1.Em4.ControlNodes".mainPnP."step".action1[250] )
      Not()
      wire#w1
      Coil( "Unit1.Em4.ControlNodes".cmAnodeMainPnP2SuctionPlateVacuum.commands.commandWorkPos )
   END_RUNG
   RUNG wire#powerrail
      I_Contact( "Unit1.Em4.ControlNodes".gaugeRnR."step".action1[1630] )
      I_Contact( "Unit1.Em4.ControlNodes".gaugeRnR."step".action1[2030] )
      Not()
   END_RUNG wire#w1
   RUNG wire#powerrail
      Contact( "Unit1.MotionNodes".PLCToMotion.Commands.StackMain.Auto )
      wire#w2
      Contact( "Unit1.EmData".PartData.EM4.anodeAlignTable.UnitData.VisionAlign.OK )
      Contact( "Unit1.MotionNodes".MotionToPLC.Status.StackMain.Busy.AutoBusy )
      Contact( "Unit1.MotionNodes".MotionToPLC.Status.OutputBits.AnodePnP2Suction )
      I_Contact( "Unit1.EmData".PartData.EM4.anodeAlignTable.UnitData.VisionAlign.NG )
      I_Contact( "Unit1.EmData".PartData.EM5.cathodeAlignTable.UnitData.VisionAlign.NG )
      I_Contact( "Unit1.EmData".PartData.EM6.stackTable.UnitData.VisionGap.NG )
   END_RUNG wire#w1
   RUNG wire#powerrail
      Contact( "Unit1.EmNodes".motionInterface.StackMain.StopMotion )
   END_RUNG wire#w2
   // the same network as SCL:
   "Unit1.Em4.ControlNodes".cm.Interlock.anodeMainPnP2SuctionPlateVacuum.work := TRUE;
   "Unit1.Em4.ControlNodes".cmAnodeMainPnP2SuctionPlateVacuum.commands.commandWorkPos := NOT (NOT "Unit1.Em4.ControlNodes".mainPnP."step".action1[1020] AND NOT "Unit1.Em4.ControlNodes".mainPnP."step".action1[118] AND NOT "Unit1.Em4.ControlNodes".mainPnP."step".action1[137] AND NOT "Unit1.Em4.ControlNodes".mainPnP."step".action1[133] AND NOT "Unit1.Em4.ControlNodes".mainPnP."step".action1[153] AND NOT "Unit1.Em4.ControlNodes".mainPnP."step".action1[250]) OR NOT (NOT "Unit1.Em4.ControlNodes".gaugeRnR."step".action1[1630] AND NOT "Unit1.Em4.ControlNodes".gaugeRnR."step".action1[2030]) OR (("Unit1.MotionNodes".PLCToMotion.Commands.StackMain.Auto OR "Unit1.EmNodes".motionInterface.StackMain.StopMotion) AND "Unit1.EmData".PartData.EM4.anodeAlignTable.UnitData.VisionAlign.OK AND "Unit1.MotionNodes".MotionToPLC.Status.StackMain.Busy.AutoBusy AND "Unit1.MotionNodes".MotionToPLC.Status.OutputBits.AnodePnP2Suction AND NOT "Unit1.EmData".PartData.EM4.anodeAlignTable.UnitData.VisionAlign.NG AND NOT "Unit1.EmData".PartData.EM5.cathodeAlignTable.UnitData.VisionAlign.NG AND NOT "Unit1.EmData".PartData.EM6.stackTable.UnitData.VisionGap.NG);
END_REGION

REGION Network 237: Call instCmAnodeMainPnP2SuctionPlateVacuum
   RUNG wire#powerrail
      #instCmAnodeMainPnP2ndSuctionPlateVacuum(feedbackHomePos := wire#w1, feedbackWorkPos := wire#w2, enable := TRUE, parentReferenceDesignator := "Unit1.Em4.Config".em.referenceDesignator.combined, enableManualCmds := #statEnableManualCmds, interlockWorkPos := "Unit1.Em4.ControlNodes".cm.Interlock.anodeMainPnP2SuctionPlateVacuum.work, interlockHomePos := "Unit1.Em4.ControlNodes".cm.Interlock.anodeMainPnP2SuctionPlateVacuum.home, configuration := "Unit1.Em4.Config".cmAnodeMainPnP2SuctionPlateVacuum, moduleInterface := "Unit1.Em4.HmiInterface".cmAnodeMainPnP2SuctionPlateVacuum, controlNode := "Unit1.Em4.ControlNodes".cmAnodeMainPnP2SuctionPlateVacuum, goToHomePos =>, goToWorkPos =>)
   END_RUNG
   RUNG wire#powerrail
      I_Contact( "BA030AZSBK06.04" )
   END_RUNG wire#w1
   RUNG wire#powerrail
      Contact( "BA030AZSBK06.04" )
   END_RUNG wire#w2
   RUNG wire#powerrail
      Contact( #instCmAnodeMainPnP2ndSuctionPlateVacuum.goToHomePos )
      I_Contact( #statUnitStatus.specialFunctions.dryRun )
      Coil( "BA030AZSBK31.03" )
   END_RUNG
   RUNG wire#powerrail
      Contact( #instCmAnodeMainPnP2ndSuctionPlateVacuum.goToWorkPos )
      I_Contact( #statUnitStatus.specialFunctions.dryRun )
      Coil( "BA030AZSBK31.02" )
   END_RUNG
   // the same network as SCL:
   #instCmAnodeMainPnP2ndSuctionPlateVacuum(enable := TRUE,   // "LBC_TwoWayActuatorCn"
                           parentReferenceDesignator := "Unit1.Em4.Config".em.referenceDesignator.combined,
                           feedbackHomePos := NOT "BA030AZSBK06.04",
                           feedbackWorkPos := "BA030AZSBK06.04",
                           enableManualCmds := #statEnableManualCmds,
                           interlockWorkPos := "Unit1.Em4.ControlNodes".cm.Interlock.anodeMainPnP2SuctionPlateVacuum.work,
                           interlockHomePos := "Unit1.Em4.ControlNodes".cm.Interlock.anodeMainPnP2SuctionPlateVacuum.home,
                           configuration := "Unit1.Em4.Config".cmAnodeMainPnP2SuctionPlateVacuum,
                           moduleInterface := "Unit1.Em4.HmiInterface".cmAnodeMainPnP2SuctionPlateVacuum,
                           controlNode := "Unit1.Em4.ControlNodes".cmAnodeMainPnP2SuctionPlateVacuum);
   "BA030AZSBK31.03" := #instCmAnodeMainPnP2ndSuctionPlateVacuum.goToHomePos AND NOT #statUnitStatus.specialFunctions.dryRun;
   "BA030AZSBK31.02" := #instCmAnodeMainPnP2ndSuctionPlateVacuum.goToWorkPos AND NOT #statUnitStatus.specialFunctions.dryRun;
END_REGION

REGION Network 239: CmAnodeAlignTableSuctionPlateVacuum Home
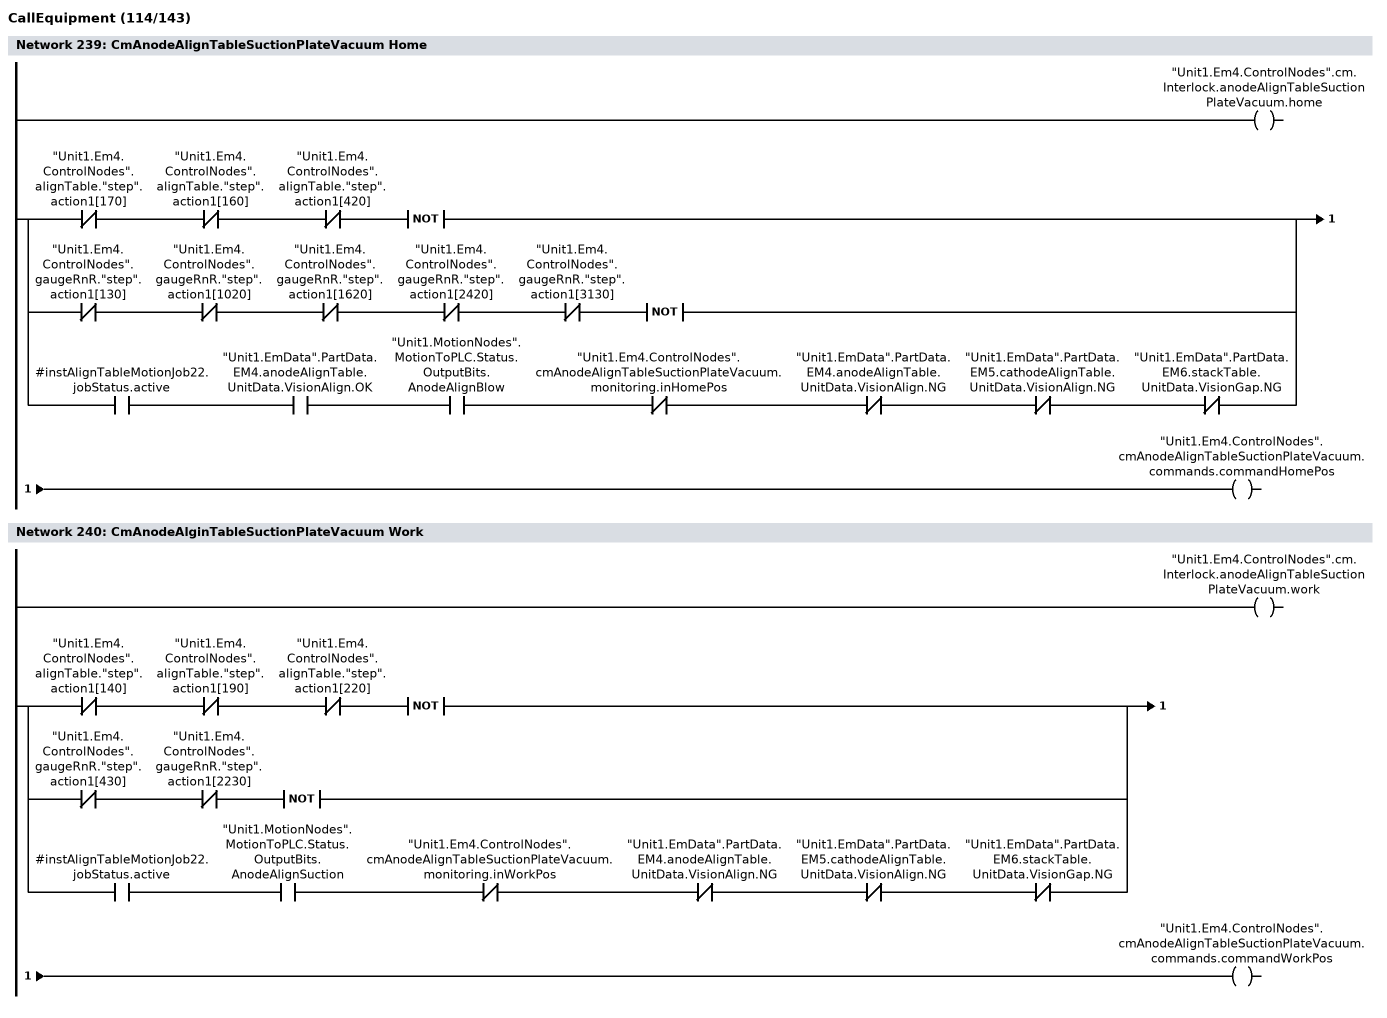
   RUNG wire#powerrail
      Coil( "Unit1.Em4.ControlNodes".cm.Interlock.anodeAlignTableSuctionPlateVacuum.home )
   END_RUNG
   RUNG wire#powerrail
      I_Contact( "Unit1.Em4.ControlNodes".alignTable."step".action1[170] )
      I_Contact( "Unit1.Em4.ControlNodes".alignTable."step".action1[160] )
      I_Contact( "Unit1.Em4.ControlNodes".alignTable."step".action1[420] )
      Not()
      wire#w1
      Coil( "Unit1.Em4.ControlNodes".cmAnodeAlignTableSuctionPlateVacuum.commands.commandHomePos )
   END_RUNG
   RUNG wire#powerrail
      I_Contact( "Unit1.Em4.ControlNodes".gaugeRnR."step".action1[130] )
      I_Contact( "Unit1.Em4.ControlNodes".gaugeRnR."step".action1[1020] )
      I_Contact( "Unit1.Em4.ControlNodes".gaugeRnR."step".action1[1620] )
      I_Contact( "Unit1.Em4.ControlNodes".gaugeRnR."step".action1[2420] )
      I_Contact( "Unit1.Em4.ControlNodes".gaugeRnR."step".action1[3130] )
      Not()
   END_RUNG wire#w1
   RUNG wire#powerrail
      Contact( #instAlignTableMotionJob22.jobStatus.active )
      Contact( "Unit1.EmData".PartData.EM4.anodeAlignTable.UnitData.VisionAlign.OK )
      Contact( "Unit1.MotionNodes".MotionToPLC.Status.OutputBits.AnodeAlignBlow )
      I_Contact( "Unit1.Em4.ControlNodes".cmAnodeAlignTableSuctionPlateVacuum.monitoring.inHomePos )
      I_Contact( "Unit1.EmData".PartData.EM4.anodeAlignTable.UnitData.VisionAlign.NG )
      I_Contact( "Unit1.EmData".PartData.EM5.cathodeAlignTable.UnitData.VisionAlign.NG )
      I_Contact( "Unit1.EmData".PartData.EM6.stackTable.UnitData.VisionGap.NG )
   END_RUNG wire#w1
   // the same network as SCL:
   "Unit1.Em4.ControlNodes".cm.Interlock.anodeAlignTableSuctionPlateVacuum.home := TRUE;
   "Unit1.Em4.ControlNodes".cmAnodeAlignTableSuctionPlateVacuum.commands.commandHomePos := NOT (NOT "Unit1.Em4.ControlNodes".alignTable."step".action1[170] AND NOT "Unit1.Em4.ControlNodes".alignTable."step".action1[160] AND NOT "Unit1.Em4.ControlNodes".alignTable."step".action1[420]) OR NOT (NOT "Unit1.Em4.ControlNodes".gaugeRnR."step".action1[130] AND NOT "Unit1.Em4.ControlNodes".gaugeRnR."step".action1[1020] AND NOT "Unit1.Em4.ControlNodes".gaugeRnR."step".action1[1620] AND NOT "Unit1.Em4.ControlNodes".gaugeRnR."step".action1[2420] AND NOT "Unit1.Em4.ControlNodes".gaugeRnR."step".action1[3130]) OR (#instAlignTableMotionJob22.jobStatus.active AND "Unit1.EmData".PartData.EM4.anodeAlignTable.UnitData.VisionAlign.OK AND "Unit1.MotionNodes".MotionToPLC.Status.OutputBits.AnodeAlignBlow AND NOT "Unit1.Em4.ControlNodes".cmAnodeAlignTableSuctionPlateVacuum.monitoring.inHomePos AND NOT "Unit1.EmData".PartData.EM4.anodeAlignTable.UnitData.VisionAlign.NG AND NOT "Unit1.EmData".PartData.EM5.cathodeAlignTable.UnitData.VisionAlign.NG AND NOT "Unit1.EmData".PartData.EM6.stackTable.UnitData.VisionGap.NG);
END_REGION

REGION Network 240: CmAnodeAlginTableSuctionPlateVacuum Work
   RUNG wire#powerrail
      Coil( "Unit1.Em4.ControlNodes".cm.Interlock.anodeAlignTableSuctionPlateVacuum.work )
   END_RUNG
   RUNG wire#powerrail
      I_Contact( "Unit1.Em4.ControlNodes".alignTable."step".action1[140] )
      I_Contact( "Unit1.Em4.ControlNodes".alignTable."step".action1[190] )
      I_Contact( "Unit1.Em4.ControlNodes".alignTable."step".action1[220] )
      Not()
      wire#w1
      Coil( "Unit1.Em4.ControlNodes".cmAnodeAlignTableSuctionPlateVacuum.commands.commandWorkPos )
   END_RUNG
   RUNG wire#powerrail
      I_Contact( "Unit1.Em4.ControlNodes".gaugeRnR."step".action1[430] )
      I_Contact( "Unit1.Em4.ControlNodes".gaugeRnR."step".action1[2230] )
      Not()
   END_RUNG wire#w1
   RUNG wire#powerrail
      Contact( #instAlignTableMotionJob22.jobStatus.active )
      Contact( "Unit1.MotionNodes".MotionToPLC.Status.OutputBits.AnodeAlignSuction )
      I_Contact( "Unit1.Em4.ControlNodes".cmAnodeAlignTableSuctionPlateVacuum.monitoring.inWorkPos )
      I_Contact( "Unit1.EmData".PartData.EM4.anodeAlignTable.UnitData.VisionAlign.NG )
      I_Contact( "Unit1.EmData".PartData.EM5.cathodeAlignTable.UnitData.VisionAlign.NG )
      I_Contact( "Unit1.EmData".PartData.EM6.stackTable.UnitData.VisionGap.NG )
   END_RUNG wire#w1
   // the same network as SCL:
   "Unit1.Em4.ControlNodes".cm.Interlock.anodeAlignTableSuctionPlateVacuum.work := TRUE;
   "Unit1.Em4.ControlNodes".cmAnodeAlignTableSuctionPlateVacuum.commands.commandWorkPos := NOT (NOT "Unit1.Em4.ControlNodes".alignTable."step".action1[140] AND NOT "Unit1.Em4.ControlNodes".alignTable."step".action1[190] AND NOT "Unit1.Em4.ControlNodes".alignTable."step".action1[220]) OR NOT (NOT "Unit1.Em4.ControlNodes".gaugeRnR."step".action1[430] AND NOT "Unit1.Em4.ControlNodes".gaugeRnR."step".action1[2230]) OR (#instAlignTableMotionJob22.jobStatus.active AND "Unit1.MotionNodes".MotionToPLC.Status.OutputBits.AnodeAlignSuction AND NOT "Unit1.Em4.ControlNodes".cmAnodeAlignTableSuctionPlateVacuum.monitoring.inWorkPos AND NOT "Unit1.EmData".PartData.EM4.anodeAlignTable.UnitData.VisionAlign.NG AND NOT "Unit1.EmData".PartData.EM5.cathodeAlignTable.UnitData.VisionAlign.NG AND NOT "Unit1.EmData".PartData.EM6.stackTable.UnitData.VisionGap.NG);
END_REGION

REGION Network 241: Call instCmAnodeAlignTalbeSuctionPlateVacuum
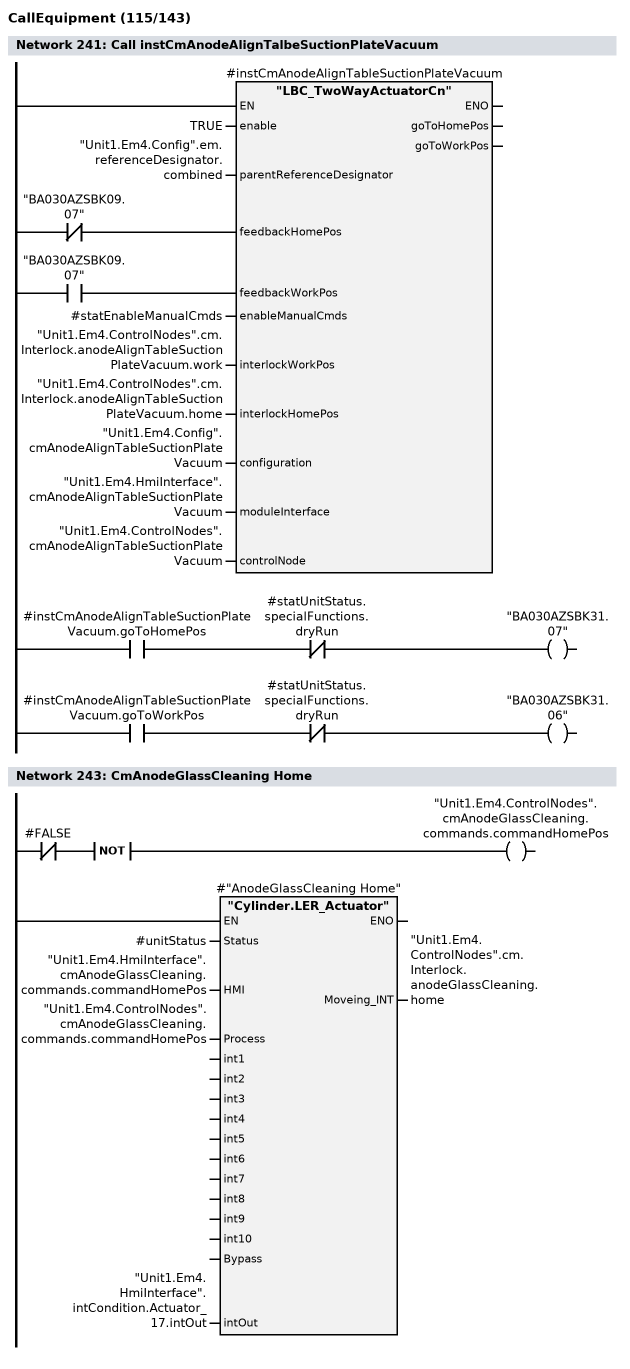
   RUNG wire#powerrail
      #instCmAnodeAlignTableSuctionPlateVacuum(feedbackHomePos := wire#w1, feedbackWorkPos := wire#w2, enable := TRUE, parentReferenceDesignator := "Unit1.Em4.Config".em.referenceDesignator.combined, enableManualCmds := #statEnableManualCmds, interlockWorkPos := "Unit1.Em4.ControlNodes".cm.Interlock.anodeAlignTableSuctionPlateVacuum.work, interlockHomePos := "Unit1.Em4.ControlNodes".cm.Interlock.anodeAlignTableSuctionPlateVacuum.home, configuration := "Unit1.Em4.Config".cmAnodeAlignTableSuctionPlateVacuum, moduleInterface := "Unit1.Em4.HmiInterface".cmAnodeAlignTableSuctionPlateVacuum, controlNode := "Unit1.Em4.ControlNodes".cmAnodeAlignTableSuctionPlateVacuum, goToHomePos =>, goToWorkPos =>)
   END_RUNG
   RUNG wire#powerrail
      I_Contact( "BA030AZSBK09.07" )
   END_RUNG wire#w1
   RUNG wire#powerrail
      Contact( "BA030AZSBK09.07" )
   END_RUNG wire#w2
   RUNG wire#powerrail
      Contact( #instCmAnodeAlignTableSuctionPlateVacuum.goToHomePos )
      I_Contact( #statUnitStatus.specialFunctions.dryRun )
      Coil( "BA030AZSBK31.07" )
   END_RUNG
   RUNG wire#powerrail
      Contact( #instCmAnodeAlignTableSuctionPlateVacuum.goToWorkPos )
      I_Contact( #statUnitStatus.specialFunctions.dryRun )
      Coil( "BA030AZSBK31.06" )
   END_RUNG
   // the same network as SCL:
   #instCmAnodeAlignTableSuctionPlateVacuum(enable := TRUE,   // "LBC_TwoWayActuatorCn"
                           parentReferenceDesignator := "Unit1.Em4.Config".em.referenceDesignator.combined,
                           feedbackHomePos := NOT "BA030AZSBK09.07",
                           feedbackWorkPos := "BA030AZSBK09.07",
                           enableManualCmds := #statEnableManualCmds,
                           interlockWorkPos := "Unit1.Em4.ControlNodes".cm.Interlock.anodeAlignTableSuctionPlateVacuum.work,
                           interlockHomePos := "Unit1.Em4.ControlNodes".cm.Interlock.anodeAlignTableSuctionPlateVacuum.home,
                           configuration := "Unit1.Em4.Config".cmAnodeAlignTableSuctionPlateVacuum,
                           moduleInterface := "Unit1.Em4.HmiInterface".cmAnodeAlignTableSuctionPlateVacuum,
                           controlNode := "Unit1.Em4.ControlNodes".cmAnodeAlignTableSuctionPlateVacuum);
   "BA030AZSBK31.07" := #instCmAnodeAlignTableSuctionPlateVacuum.goToHomePos AND NOT #statUnitStatus.specialFunctions.dryRun;
   "BA030AZSBK31.06" := #instCmAnodeAlignTableSuctionPlateVacuum.goToWorkPos AND NOT #statUnitStatus.specialFunctions.dryRun;
END_REGION

REGION Network 243: CmAnodeGlassCleaning Home
   RUNG wire#powerrail
      I_Contact( #FALSE )
      Not()
      Coil( "Unit1.Em4.ControlNodes".cmAnodeGlassCleaning.commands.commandHomePos )
   END_RUNG
   RUNG wire#powerrail
      #"AnodeGlassCleaning Home"(Status := #unitStatus, HMI := "Unit1.Em4.HmiInterface".cmAnodeGlassCleaning.commands.commandHomePos, Process := "Unit1.Em4.ControlNodes".cmAnodeGlassCleaning.commands.commandHomePos, int1 :=, int2 :=, int3 :=, int4 :=, int5 :=, int6 :=, int7 :=, int8 :=, int9 :=, int10 :=, Bypass :=, intOut := "Unit1.Em4.HmiInterface".intCondition.Actuator_17.intOut, Moveing_INT => "Unit1.Em4.ControlNodes".cm.Interlock.anodeGlassCleaning.home)
   END_RUNG
   // the same network as SCL:
   "Unit1.Em4.ControlNodes".cmAnodeGlassCleaning.commands.commandHomePos := NOT (NOT #FALSE);
   #"AnodeGlassCleaning Home"(Status := #unitStatus,   // "Cylinder.LER_Actuator"
                           HMI := "Unit1.Em4.HmiInterface".cmAnodeGlassCleaning.commands.commandHomePos,
                           Process := "Unit1.Em4.ControlNodes".cmAnodeGlassCleaning.commands.commandHomePos,
                           intOut := "Unit1.Em4.HmiInterface".intCondition.Actuator_17.intOut,
                           Moveing_INT => "Unit1.Em4.ControlNodes".cm.Interlock.anodeGlassCleaning.home);
END_REGION

REGION Network 244: CmAnodeGlassCleaning Work
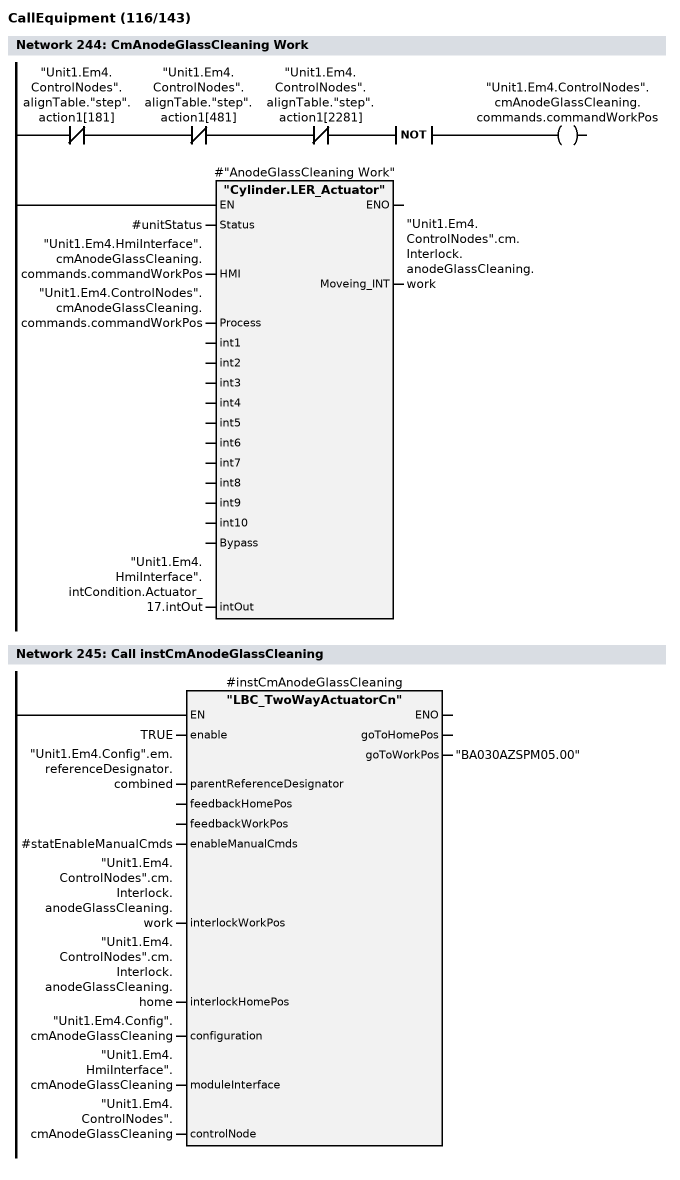
   RUNG wire#powerrail
      I_Contact( "Unit1.Em4.ControlNodes".alignTable."step".action1[181] )
      I_Contact( "Unit1.Em4.ControlNodes".alignTable."step".action1[481] )
      I_Contact( "Unit1.Em4.ControlNodes".alignTable."step".action1[2281] )
      Not()
      Coil( "Unit1.Em4.ControlNodes".cmAnodeGlassCleaning.commands.commandWorkPos )
   END_RUNG
   RUNG wire#powerrail
      #"AnodeGlassCleaning Work"(Status := #unitStatus, HMI := "Unit1.Em4.HmiInterface".cmAnodeGlassCleaning.commands.commandWorkPos, Process := "Unit1.Em4.ControlNodes".cmAnodeGlassCleaning.commands.commandWorkPos, int1 :=, int2 :=, int3 :=, int4 :=, int5 :=, int6 :=, int7 :=, int8 :=, int9 :=, int10 :=, Bypass :=, intOut := "Unit1.Em4.HmiInterface".intCondition.Actuator_17.intOut, Moveing_INT => "Unit1.Em4.ControlNodes".cm.Interlock.anodeGlassCleaning.work)
   END_RUNG
   // the same network as SCL:
   "Unit1.Em4.ControlNodes".cmAnodeGlassCleaning.commands.commandWorkPos := NOT (NOT "Unit1.Em4.ControlNodes".alignTable."step".action1[181] AND NOT "Unit1.Em4.ControlNodes".alignTable."step".action1[481] AND NOT "Unit1.Em4.ControlNodes".alignTable."step".action1[2281]);
   #"AnodeGlassCleaning Work"(Status := #unitStatus,   // "Cylinder.LER_Actuator"
                           HMI := "Unit1.Em4.HmiInterface".cmAnodeGlassCleaning.commands.commandWorkPos,
                           Process := "Unit1.Em4.ControlNodes".cmAnodeGlassCleaning.commands.commandWorkPos,
                           intOut := "Unit1.Em4.HmiInterface".intCondition.Actuator_17.intOut,
                           Moveing_INT => "Unit1.Em4.ControlNodes".cm.Interlock.anodeGlassCleaning.work);
END_REGION

REGION Network 245: Call instCmAnodeGlassCleaning
   RUNG wire#powerrail
      #instCmAnodeGlassCleaning(enable := TRUE, parentReferenceDesignator := "Unit1.Em4.Config".em.referenceDesignator.combined, feedbackHomePos :=, feedbackWorkPos :=, enableManualCmds := #statEnableManualCmds, interlockWorkPos := "Unit1.Em4.ControlNodes".cm.Interlock.anodeGlassCleaning.work, interlockHomePos := "Unit1.Em4.ControlNodes".cm.Interlock.anodeGlassCleaning.home, configuration := "Unit1.Em4.Config".cmAnodeGlassCleaning, moduleInterface := "Unit1.Em4.HmiInterface".cmAnodeGlassCleaning, controlNode := "Unit1.Em4.ControlNodes".cmAnodeGlassCleaning, goToHomePos =>, goToWorkPos => "BA030AZSPM05.00")
   END_RUNG
   // the same network as SCL:
   #instCmAnodeGlassCleaning(enable := TRUE,   // "LBC_TwoWayActuatorCn"
                           parentReferenceDesignator := "Unit1.Em4.Config".em.referenceDesignator.combined,
                           enableManualCmds := #statEnableManualCmds,
                           interlockWorkPos := "Unit1.Em4.ControlNodes".cm.Interlock.anodeGlassCleaning.work,
                           interlockHomePos := "Unit1.Em4.ControlNodes".cm.Interlock.anodeGlassCleaning.home,
                           configuration := "Unit1.Em4.Config".cmAnodeGlassCleaning,
                           moduleInterface := "Unit1.Em4.HmiInterface".cmAnodeGlassCleaning,
                           controlNode := "Unit1.Em4.ControlNodes".cmAnodeGlassCleaning,
                           goToWorkPos => "BA030AZSPM05.00");
END_REGION

REGION Network 247: CmAnodeNgPnpUpDown Home
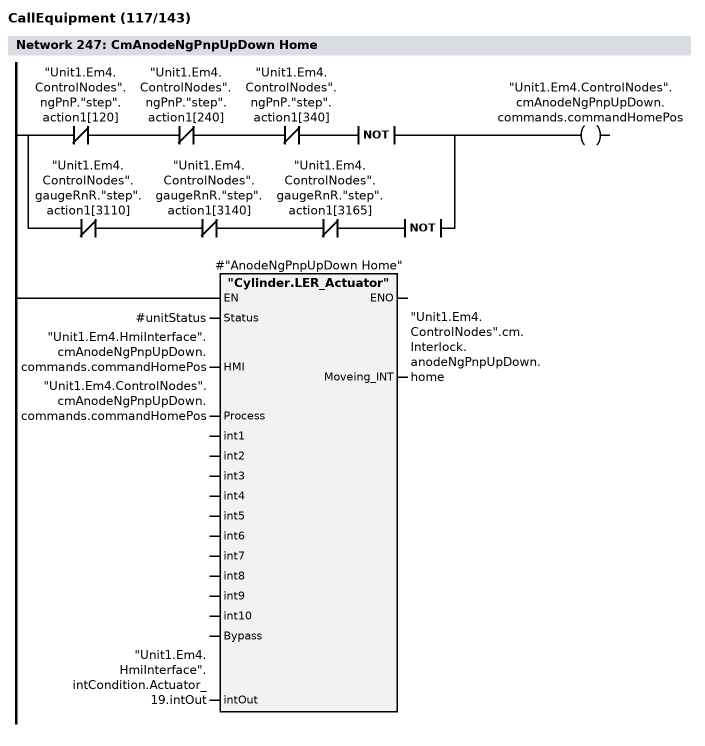
   RUNG wire#powerrail
      I_Contact( "Unit1.Em4.ControlNodes".ngPnP."step".action1[120] )
      I_Contact( "Unit1.Em4.ControlNodes".ngPnP."step".action1[240] )
      I_Contact( "Unit1.Em4.ControlNodes".ngPnP."step".action1[340] )
      Not()
      wire#w1
      Coil( "Unit1.Em4.ControlNodes".cmAnodeNgPnpUpDown.commands.commandHomePos )
   END_RUNG
   RUNG wire#powerrail
      I_Contact( "Unit1.Em4.ControlNodes".gaugeRnR."step".action1[3110] )
      I_Contact( "Unit1.Em4.ControlNodes".gaugeRnR."step".action1[3140] )
      I_Contact( "Unit1.Em4.ControlNodes".gaugeRnR."step".action1[3165] )
      Not()
   END_RUNG wire#w1
   RUNG wire#powerrail
      #"AnodeNgPnpUpDown Home"(Status := #unitStatus, HMI := "Unit1.Em4.HmiInterface".cmAnodeNgPnpUpDown.commands.commandHomePos, Process := "Unit1.Em4.ControlNodes".cmAnodeNgPnpUpDown.commands.commandHomePos, int1 :=, int2 :=, int3 :=, int4 :=, int5 :=, int6 :=, int7 :=, int8 :=, int9 :=, int10 :=, Bypass :=, intOut := "Unit1.Em4.HmiInterface".intCondition.Actuator_19.intOut, Moveing_INT => "Unit1.Em4.ControlNodes".cm.Interlock.anodeNgPnpUpDown.home)
   END_RUNG
   // the same network as SCL:
   "Unit1.Em4.ControlNodes".cmAnodeNgPnpUpDown.commands.commandHomePos := NOT (NOT "Unit1.Em4.ControlNodes".ngPnP."step".action1[120] AND NOT "Unit1.Em4.ControlNodes".ngPnP."step".action1[240] AND NOT "Unit1.Em4.ControlNodes".ngPnP."step".action1[340]) OR NOT (NOT "Unit1.Em4.ControlNodes".gaugeRnR."step".action1[3110] AND NOT "Unit1.Em4.ControlNodes".gaugeRnR."step".action1[3140] AND NOT "Unit1.Em4.ControlNodes".gaugeRnR."step".action1[3165]);
   #"AnodeNgPnpUpDown Home"(Status := #unitStatus,   // "Cylinder.LER_Actuator"
                           HMI := "Unit1.Em4.HmiInterface".cmAnodeNgPnpUpDown.commands.commandHomePos,
                           Process := "Unit1.Em4.ControlNodes".cmAnodeNgPnpUpDown.commands.commandHomePos,
                           intOut := "Unit1.Em4.HmiInterface".intCondition.Actuator_19.intOut,
                           Moveing_INT => "Unit1.Em4.ControlNodes".cm.Interlock.anodeNgPnpUpDown.home);
END_REGION

REGION Network 248: CmAnodeNgPnpUpDown Work
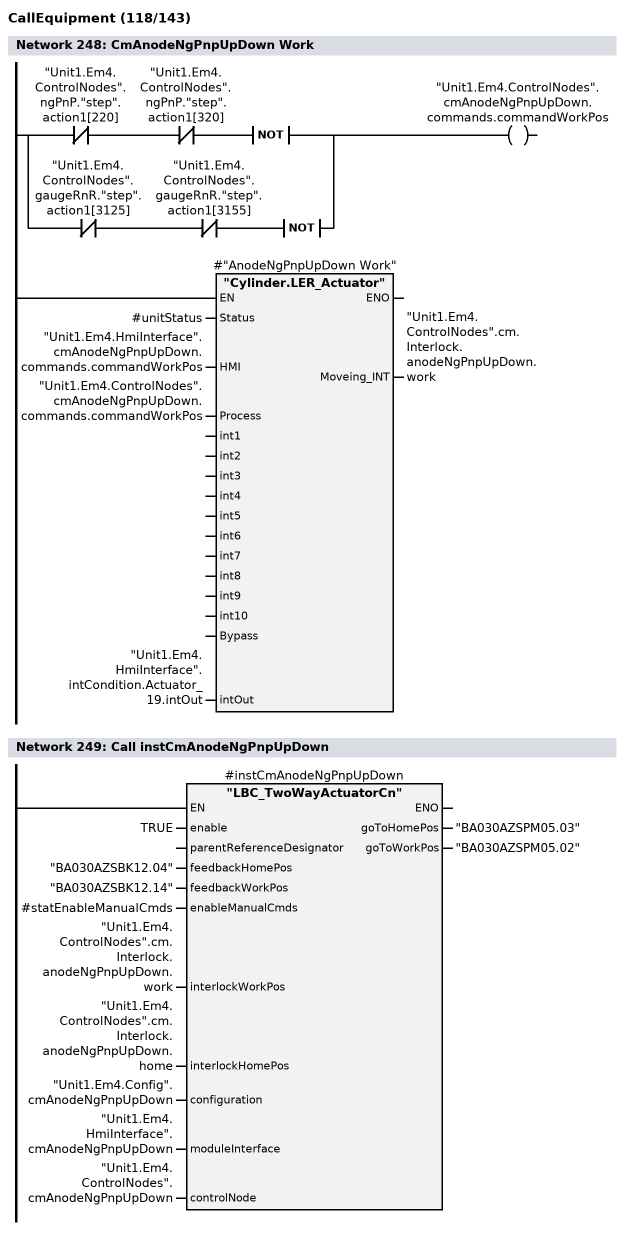
   RUNG wire#powerrail
      I_Contact( "Unit1.Em4.ControlNodes".ngPnP."step".action1[220] )
      I_Contact( "Unit1.Em4.ControlNodes".ngPnP."step".action1[320] )
      Not()
      wire#w1
      Coil( "Unit1.Em4.ControlNodes".cmAnodeNgPnpUpDown.commands.commandWorkPos )
   END_RUNG
   RUNG wire#powerrail
      I_Contact( "Unit1.Em4.ControlNodes".gaugeRnR."step".action1[3125] )
      I_Contact( "Unit1.Em4.ControlNodes".gaugeRnR."step".action1[3155] )
      Not()
   END_RUNG wire#w1
   RUNG wire#powerrail
      #"AnodeNgPnpUpDown Work"(Status := #unitStatus, HMI := "Unit1.Em4.HmiInterface".cmAnodeNgPnpUpDown.commands.commandWorkPos, Process := "Unit1.Em4.ControlNodes".cmAnodeNgPnpUpDown.commands.commandWorkPos, int1 :=, int2 :=, int3 :=, int4 :=, int5 :=, int6 :=, int7 :=, int8 :=, int9 :=, int10 :=, Bypass :=, intOut := "Unit1.Em4.HmiInterface".intCondition.Actuator_19.intOut, Moveing_INT => "Unit1.Em4.ControlNodes".cm.Interlock.anodeNgPnpUpDown.work)
   END_RUNG
   // the same network as SCL:
   "Unit1.Em4.ControlNodes".cmAnodeNgPnpUpDown.commands.commandWorkPos := NOT (NOT "Unit1.Em4.ControlNodes".ngPnP."step".action1[220] AND NOT "Unit1.Em4.ControlNodes".ngPnP."step".action1[320]) OR NOT (NOT "Unit1.Em4.ControlNodes".gaugeRnR."step".action1[3125] AND NOT "Unit1.Em4.ControlNodes".gaugeRnR."step".action1[3155]);
   #"AnodeNgPnpUpDown Work"(Status := #unitStatus,   // "Cylinder.LER_Actuator"
                           HMI := "Unit1.Em4.HmiInterface".cmAnodeNgPnpUpDown.commands.commandWorkPos,
                           Process := "Unit1.Em4.ControlNodes".cmAnodeNgPnpUpDown.commands.commandWorkPos,
                           intOut := "Unit1.Em4.HmiInterface".intCondition.Actuator_19.intOut,
                           Moveing_INT => "Unit1.Em4.ControlNodes".cm.Interlock.anodeNgPnpUpDown.work);
END_REGION

REGION Network 249: Call instCmAnodeNgPnpUpDown
   RUNG wire#powerrail
      #instCmAnodeNgPnpUpDown(enable := TRUE, parentReferenceDesignator :=, feedbackHomePos := "BA030AZSBK12.04", feedbackWorkPos := "BA030AZSBK12.14", enableManualCmds := #statEnableManualCmds, interlockWorkPos := "Unit1.Em4.ControlNodes".cm.Interlock.anodeNgPnpUpDown.work, interlockHomePos := "Unit1.Em4.ControlNodes".cm.Interlock.anodeNgPnpUpDown.home, configuration := "Unit1.Em4.Config".cmAnodeNgPnpUpDown, moduleInterface := "Unit1.Em4.HmiInterface".cmAnodeNgPnpUpDown, controlNode := "Unit1.Em4.ControlNodes".cmAnodeNgPnpUpDown, goToHomePos => "BA030AZSPM05.03", goToWorkPos => "BA030AZSPM05.02")
   END_RUNG
   // the same network as SCL:
   #instCmAnodeNgPnpUpDown(enable := TRUE,   // "LBC_TwoWayActuatorCn"
                           feedbackHomePos := "BA030AZSBK12.04",
                           feedbackWorkPos := "BA030AZSBK12.14",
                           enableManualCmds := #statEnableManualCmds,
                           interlockWorkPos := "Unit1.Em4.ControlNodes".cm.Interlock.anodeNgPnpUpDown.work,
                           interlockHomePos := "Unit1.Em4.ControlNodes".cm.Interlock.anodeNgPnpUpDown.home,
                           configuration := "Unit1.Em4.Config".cmAnodeNgPnpUpDown,
                           moduleInterface := "Unit1.Em4.HmiInterface".cmAnodeNgPnpUpDown,
                           controlNode := "Unit1.Em4.ControlNodes".cmAnodeNgPnpUpDown,
                           goToHomePos => "BA030AZSPM05.03",
                           goToWorkPos => "BA030AZSPM05.02");
END_REGION

REGION Network 251: CmAnodeNgPnp1stFwdBwd Home
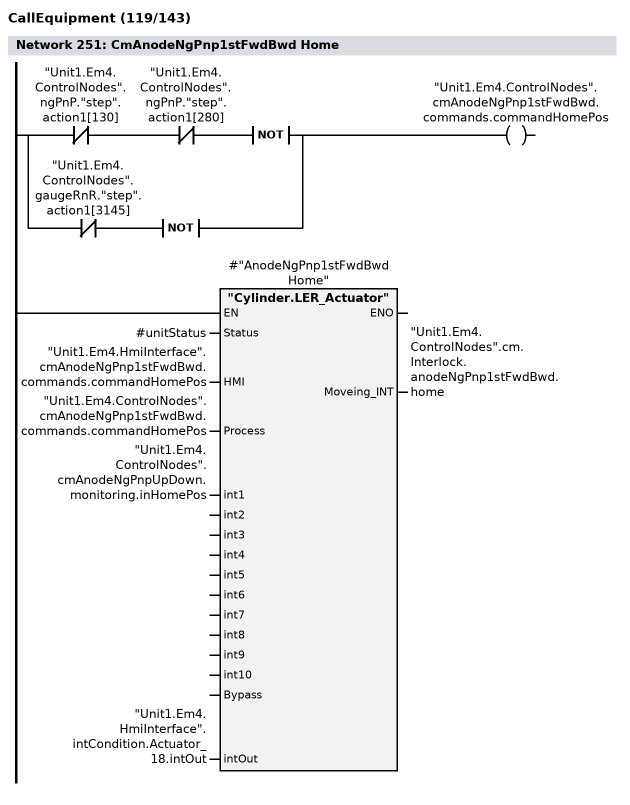
   RUNG wire#powerrail
      I_Contact( "Unit1.Em4.ControlNodes".ngPnP."step".action1[130] )
      I_Contact( "Unit1.Em4.ControlNodes".ngPnP."step".action1[280] )
      Not()
      wire#w1
      Coil( "Unit1.Em4.ControlNodes".cmAnodeNgPnp1stFwdBwd.commands.commandHomePos )
   END_RUNG
   RUNG wire#powerrail
      I_Contact( "Unit1.Em4.ControlNodes".gaugeRnR."step".action1[3145] )
      Not()
   END_RUNG wire#w1
   RUNG wire#powerrail
      #"AnodeNgPnp1stFwdBwd Home"(Status := #unitStatus, HMI := "Unit1.Em4.HmiInterface".cmAnodeNgPnp1stFwdBwd.commands.commandHomePos, Process := "Unit1.Em4.ControlNodes".cmAnodeNgPnp1stFwdBwd.commands.commandHomePos, int1 := "Unit1.Em4.ControlNodes".cmAnodeNgPnpUpDown.monitoring.inHomePos, int2 :=, int3 :=, int4 :=, int5 :=, int6 :=, int7 :=, int8 :=, int9 :=, int10 :=, Bypass :=, intOut := "Unit1.Em4.HmiInterface".intCondition.Actuator_18.intOut, Moveing_INT => "Unit1.Em4.ControlNodes".cm.Interlock.anodeNgPnp1stFwdBwd.home)
   END_RUNG
   // the same network as SCL:
   "Unit1.Em4.ControlNodes".cmAnodeNgPnp1stFwdBwd.commands.commandHomePos := NOT (NOT "Unit1.Em4.ControlNodes".ngPnP."step".action1[130] AND NOT "Unit1.Em4.ControlNodes".ngPnP."step".action1[280]) OR NOT (NOT "Unit1.Em4.ControlNodes".gaugeRnR."step".action1[3145]);
   #"AnodeNgPnp1stFwdBwd Home"(Status := #unitStatus,   // "Cylinder.LER_Actuator"
                           HMI := "Unit1.Em4.HmiInterface".cmAnodeNgPnp1stFwdBwd.commands.commandHomePos,
                           Process := "Unit1.Em4.ControlNodes".cmAnodeNgPnp1stFwdBwd.commands.commandHomePos,
                           int1 := "Unit1.Em4.ControlNodes".cmAnodeNgPnpUpDown.monitoring.inHomePos,
                           intOut := "Unit1.Em4.HmiInterface".intCondition.Actuator_18.intOut,
                           Moveing_INT => "Unit1.Em4.ControlNodes".cm.Interlock.anodeNgPnp1stFwdBwd.home);
END_REGION

REGION Network 252: CmAnodeNgPnp1stFwdBwd Work
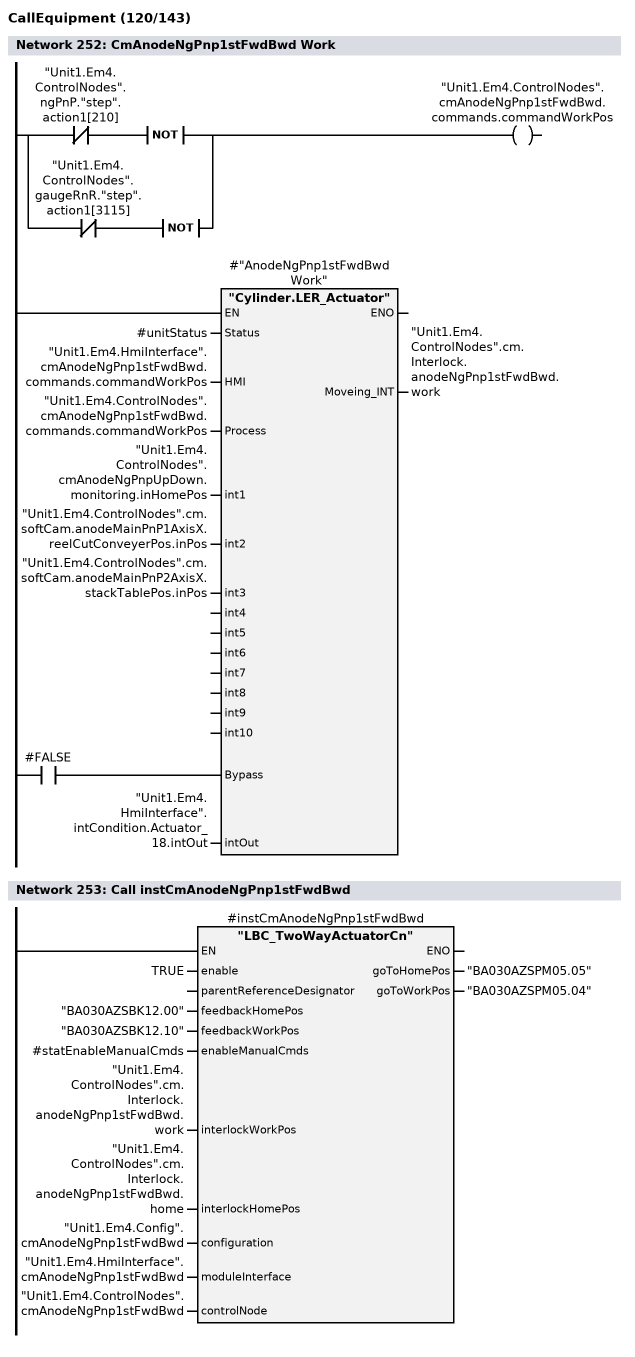
   RUNG wire#powerrail
      I_Contact( "Unit1.Em4.ControlNodes".ngPnP."step".action1[210] )
      Not()
      wire#w1
      Coil( "Unit1.Em4.ControlNodes".cmAnodeNgPnp1stFwdBwd.commands.commandWorkPos )
   END_RUNG
   RUNG wire#powerrail
      I_Contact( "Unit1.Em4.ControlNodes".gaugeRnR."step".action1[3115] )
      Not()
   END_RUNG wire#w1
   RUNG wire#powerrail
      #"AnodeNgPnp1stFwdBwd Work"(Bypass := wire#w2, Status := #unitStatus, HMI := "Unit1.Em4.HmiInterface".cmAnodeNgPnp1stFwdBwd.commands.commandWorkPos, Process := "Unit1.Em4.ControlNodes".cmAnodeNgPnp1stFwdBwd.commands.commandWorkPos, int1 := "Unit1.Em4.ControlNodes".cmAnodeNgPnpUpDown.monitoring.inHomePos, int2 := "Unit1.Em4.ControlNodes".cm.softCam.anodeMainPnP1AxisX.reelCutConveyerPos.inPos, int3 := "Unit1.Em4.ControlNodes".cm.softCam.anodeMainPnP2AxisX.stackTablePos.inPos, int4 :=, int5 :=, int6 :=, int7 :=, int8 :=, int9 :=, int10 :=, intOut := "Unit1.Em4.HmiInterface".intCondition.Actuator_18.intOut, Moveing_INT => "Unit1.Em4.ControlNodes".cm.Interlock.anodeNgPnp1stFwdBwd.work)
   END_RUNG
   RUNG wire#powerrail
      Contact( #FALSE )
   END_RUNG wire#w2
   // the same network as SCL:
   "Unit1.Em4.ControlNodes".cmAnodeNgPnp1stFwdBwd.commands.commandWorkPos := NOT (NOT "Unit1.Em4.ControlNodes".ngPnP."step".action1[210]) OR NOT (NOT "Unit1.Em4.ControlNodes".gaugeRnR."step".action1[3115]);
   #"AnodeNgPnp1stFwdBwd Work"(Status := #unitStatus,   // "Cylinder.LER_Actuator"
                           HMI := "Unit1.Em4.HmiInterface".cmAnodeNgPnp1stFwdBwd.commands.commandWorkPos,
                           Process := "Unit1.Em4.ControlNodes".cmAnodeNgPnp1stFwdBwd.commands.commandWorkPos,
                           int1 := "Unit1.Em4.ControlNodes".cmAnodeNgPnpUpDown.monitoring.inHomePos,
                           int2 := "Unit1.Em4.ControlNodes".cm.softCam.anodeMainPnP1AxisX.reelCutConveyerPos.inPos,
                           int3 := "Unit1.Em4.ControlNodes".cm.softCam.anodeMainPnP2AxisX.stackTablePos.inPos,
                           Bypass := #FALSE,
                           intOut := "Unit1.Em4.HmiInterface".intCondition.Actuator_18.intOut,
                           Moveing_INT => "Unit1.Em4.ControlNodes".cm.Interlock.anodeNgPnp1stFwdBwd.work);
END_REGION

REGION Network 253: Call instCmAnodeNgPnp1stFwdBwd
   RUNG wire#powerrail
      #instCmAnodeNgPnp1stFwdBwd(enable := TRUE, parentReferenceDesignator :=, feedbackHomePos := "BA030AZSBK12.00", feedbackWorkPos := "BA030AZSBK12.10", enableManualCmds := #statEnableManualCmds, interlockWorkPos := "Unit1.Em4.ControlNodes".cm.Interlock.anodeNgPnp1stFwdBwd.work, interlockHomePos := "Unit1.Em4.ControlNodes".cm.Interlock.anodeNgPnp1stFwdBwd.home, configuration := "Unit1.Em4.Config".cmAnodeNgPnp1stFwdBwd, moduleInterface := "Unit1.Em4.HmiInterface".cmAnodeNgPnp1stFwdBwd, controlNode := "Unit1.Em4.ControlNodes".cmAnodeNgPnp1stFwdBwd, goToHomePos => "BA030AZSPM05.05", goToWorkPos => "BA030AZSPM05.04")
   END_RUNG
   // the same network as SCL:
   #instCmAnodeNgPnp1stFwdBwd(enable := TRUE,   // "LBC_TwoWayActuatorCn"
                           feedbackHomePos := "BA030AZSBK12.00",
                           feedbackWorkPos := "BA030AZSBK12.10",
                           enableManualCmds := #statEnableManualCmds,
                           interlockWorkPos := "Unit1.Em4.ControlNodes".cm.Interlock.anodeNgPnp1stFwdBwd.work,
                           interlockHomePos := "Unit1.Em4.ControlNodes".cm.Interlock.anodeNgPnp1stFwdBwd.home,
                           configuration := "Unit1.Em4.Config".cmAnodeNgPnp1stFwdBwd,
                           moduleInterface := "Unit1.Em4.HmiInterface".cmAnodeNgPnp1stFwdBwd,
                           controlNode := "Unit1.Em4.ControlNodes".cmAnodeNgPnp1stFwdBwd,
                           goToHomePos => "BA030AZSPM05.05",
                           goToWorkPos => "BA030AZSPM05.04");
END_REGION

REGION Network 255: CmAnodeNgPnp2ndFwdBwd Home
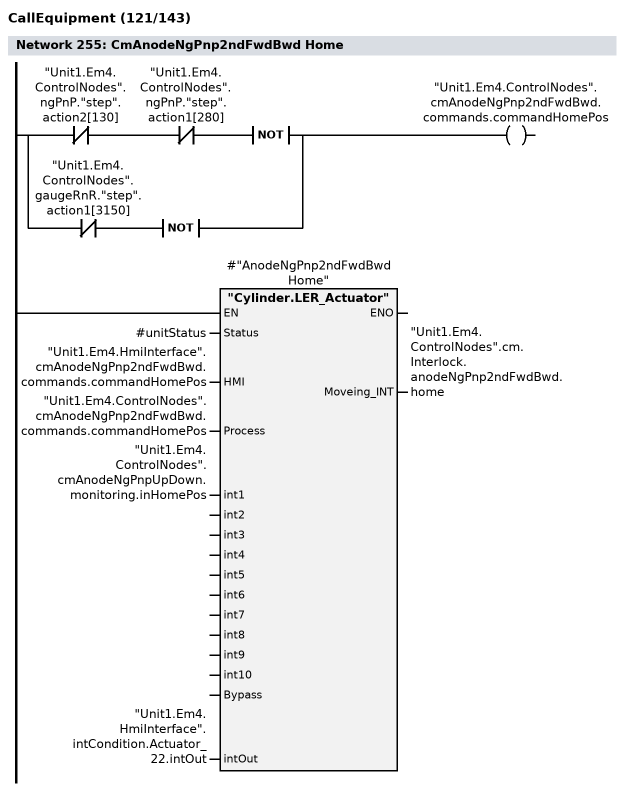
   RUNG wire#powerrail
      I_Contact( "Unit1.Em4.ControlNodes".ngPnP."step".action2[130] )
      I_Contact( "Unit1.Em4.ControlNodes".ngPnP."step".action1[280] )
      Not()
      wire#w1
      Coil( "Unit1.Em4.ControlNodes".cmAnodeNgPnp2ndFwdBwd.commands.commandHomePos )
   END_RUNG
   RUNG wire#powerrail
      I_Contact( "Unit1.Em4.ControlNodes".gaugeRnR."step".action1[3150] )
      Not()
   END_RUNG wire#w1
   RUNG wire#powerrail
      #"AnodeNgPnp2ndFwdBwd Home"(Status := #unitStatus, HMI := "Unit1.Em4.HmiInterface".cmAnodeNgPnp2ndFwdBwd.commands.commandHomePos, Process := "Unit1.Em4.ControlNodes".cmAnodeNgPnp2ndFwdBwd.commands.commandHomePos, int1 := "Unit1.Em4.ControlNodes".cmAnodeNgPnpUpDown.monitoring.inHomePos, int2 :=, int3 :=, int4 :=, int5 :=, int6 :=, int7 :=, int8 :=, int9 :=, int10 :=, Bypass :=, intOut := "Unit1.Em4.HmiInterface".intCondition.Actuator_22.intOut, Moveing_INT => "Unit1.Em4.ControlNodes".cm.Interlock.anodeNgPnp2ndFwdBwd.home)
   END_RUNG
   // the same network as SCL:
   "Unit1.Em4.ControlNodes".cmAnodeNgPnp2ndFwdBwd.commands.commandHomePos := NOT (NOT "Unit1.Em4.ControlNodes".ngPnP."step".action2[130] AND NOT "Unit1.Em4.ControlNodes".ngPnP."step".action1[280]) OR NOT (NOT "Unit1.Em4.ControlNodes".gaugeRnR."step".action1[3150]);
   #"AnodeNgPnp2ndFwdBwd Home"(Status := #unitStatus,   // "Cylinder.LER_Actuator"
                           HMI := "Unit1.Em4.HmiInterface".cmAnodeNgPnp2ndFwdBwd.commands.commandHomePos,
                           Process := "Unit1.Em4.ControlNodes".cmAnodeNgPnp2ndFwdBwd.commands.commandHomePos,
                           int1 := "Unit1.Em4.ControlNodes".cmAnodeNgPnpUpDown.monitoring.inHomePos,
                           intOut := "Unit1.Em4.HmiInterface".intCondition.Actuator_22.intOut,
                           Moveing_INT => "Unit1.Em4.ControlNodes".cm.Interlock.anodeNgPnp2ndFwdBwd.home);
END_REGION

REGION Network 256: CmAnodeNgPnp2ndFwdBwd Work
